  MoveL 642 to (10.69, 196.46, 60) mm, rotated rx -73.66 ry -11.39 rz 28.02 deg; joints [-11.348, -51.869, 112.326, 18.148, -107.646, 15.462, -1511.595]
  MoveL 643 to (4.64, 195.67, 50) mm, rotated rx -73.16 ry -13.02 rz 26.6 deg; joints [-11.489, -49.859, 112.079, 20.024, -113.289, 18.13, -1506.075]
  MoveL 644 to (-1.18, 195.49, 40) mm, rotated rx -74.98 ry -12.29 rz 16.89 deg; joints [-11.645, -52.231, 112.35, 18.85, -106.89, 14.37, -1500.872]
  MoveL 645 to (-6.67, 195.86, 30) mm, rotated rx -74.62 ry -14.16 rz 16.83 deg; joints [-11.702, -49.919, 112.059, 21.112, -113.427, 17.304, -1496.017]
  MoveL 646 to (-11.76, 196.67, 20) mm, rotated rx -76.4 ry -13.89 rz 8.51 deg; joints [-11.758, -51.951, 112.266, 20.461, -107.995, 13.792, -1491.54]
  MoveL 647 to (-16.38, 197.8, 10) mm, rotated rx -78.17 ry -13.98 rz 0.96 deg; joints [-11.742, -53.642, 112.118, 20.427, -102.896, 10.543, -1487.469]
  MoveL 648 to (-20.49, 199.16, 0) mm, rotated rx -78.17 ry -13.98 rz 0.96 deg; joints [-12.168, -53.619, 111.889, 20.096, -102.626, 10.685, -1487.469]
  Set speed (1000.0 mm/s)
  MoveL 649 to (-20.49, 199.16, 0) mm, rotated rx -78.17 ry -13.98 rz 0.96 deg; joints [-12.168, -53.619, 111.889, 20.096, -102.626, 10.685, -1487.469]
  Set speed (1000.0 mm/s)
  MoveL 650 to (37.11, 300.24, 290) mm, rotated rx -90 ry -25 rz -166.45 deg; joints [2.992, -46.004, 98.028, 40.584, -108.594, -7.061, -1313.547]
  MoveL 651 to (37.11, 300.24, 290) mm, rotated rx -90 ry -25 rz -166.45 deg; joints [2.992, -46.004, 98.028, 40.584, -108.594, -7.061, -1313.547]
  Set speed (60.0 mm/s)
  MoveL 652 to (43.85, 319.91, 290) mm, rotated rx -90 ry -25 rz -162.09 deg; joints [2.992, -46.901, 97.924, 40.37, -107.832, -7.745, -1317.907]
  Set speed (1000.0 mm/s)
  MoveL 653 to (43.85, 319.91, 290) mm, rotated rx -90 ry -25 rz -162.09 deg; joints [2.992, -46.901, 97.924, 40.37, -107.832, -7.745, -1317.907]
  Set speed (1000.0 mm/s)
  MoveL 654 to (-20.49, 199.16, 0) mm, rotated rx -90 ry -25 rz 28.05 deg; joints [-7.468, -49.938, 106.45, 34.613, -108.412, 0.917, -1148.047]
  MoveL 655 to (-20.49, 199.16, 0) mm, rotated rx -90 ry -25 rz 28.05 deg; joints [-7.468, -49.938, 106.45, 34.613, -108.412, 0.917, -1148.047]
  Set speed (60.0 mm/s)
  MoveL 656 to (-20.57, 178.36, 0) mm, rotated rx -90 ry -25 rz 33.98 deg; joints [-7.468, -50.9, 106.359, 34.42, -107.545, 0.29, -1153.977]
  Set speed (1000.0 mm/s)
  MoveL 657 to (-20.57, 178.36, 0) mm, rotated rx -90 ry -25 rz 33.98 deg; joints [-7.468, -50.9, 106.359, 34.42, -107.545, 0.29, -1153.977]
  Set speed (1000.0 mm/s)
  MoveL 658 to (-20.49, 199.16, 0) mm, rotated rx -90 ry -25 rz 28.05 deg; joints [-7.468, -49.938, 106.45, 34.613, -108.412, 0.917, -1148.047]
  MoveL 659 to (-20.49, 199.16, 0) mm, rotated rx -90 ry -25 rz 28.05 deg; joints [-7.468, -49.938, 106.45, 34.613, -108.412, 0.917, -1148.047]
  Set speed (60.0 mm/s)
  MoveL 660 to (-16.38, 197.8, 10) mm, rotated rx -90 ry -25 rz 32.58 deg; joints [-7.088, -49.83, 106.249, 34.855, -108.455, 0.679, -1152.579]
  MoveL 661 to (-11.76, 196.67, 20) mm, rotated rx -90 ry -25 rz 37.57 deg; joints [-6.709, -49.719, 106.042, 35.094, -108.496, 0.44, -1157.568]
  MoveL 662 to (-6.67, 195.86, 30) mm, rotated rx -90 ry -25 rz 42.97 deg; joints [-6.332, -49.607, 105.829, 35.331, -108.535, 0.198, -1162.975]
  MoveL 663 to (-1.18, 195.49, 40) mm, rotated rx -90 ry -25 rz 48.76 deg; joints [-5.956, -49.493, 105.609, 35.566, -108.57, -0.047, -1168.76]
  MoveL 664 to (4.64, 195.67, 50) mm, rotated rx -90 ry -25 rz 54.88 deg; joints [-5.581, -49.378, 105.383, 35.798, -108.602, -0.295, -1174.88]
  MoveL 665 to (10.69, 196.46, 60) mm, rotated rx -90 ry -25 rz 61.29 deg; joints [-5.207, -49.263, 105.151, 36.028, -108.63, -0.546, -1181.291]
  MoveL 666 to (16.86, 197.94, 70) mm, rotated rx -90 ry -25 rz 67.95 deg; joints [-4.834, -49.146, 104.912, 36.254, -108.654, -0.801, -1187.947]
  MoveL 667 to (23.03, 200.17, 80) mm, rotated rx -90 ry -25 rz 74.8 deg; joints [-4.463, -49.03, 104.666, 36.478, -108.674, -1.059, -1194.802]
  MoveL 668 to (29.06, 203.14, 90) mm, rotated rx -90 ry -25 rz 81.81 deg; joints [-4.093, -48.913, 104.414, 36.699, -108.69, -1.322, -1201.809]
  MoveL 669 to (34.83, 206.87, 100) mm, rotated rx -90 ry -25 rz 88.92 deg; joints [-3.725, -48.796, 104.156, 36.917, -108.702, -1.588, -1208.92]
  MoveL 670 to (40.19, 211.31, 110) mm, rotated rx -90 ry -25 rz 96.09 deg; joints [-3.358, -48.678, 103.891, 37.133, -108.711, -1.858, -1216.089]
  MoveL 671 to (45.04, 216.4, 120) mm, rotated rx -90 ry -25 rz 103.27 deg; joints [-2.992, -48.56, 103.619, 37.345, -108.716, -2.131, -1223.271]
  MoveL 672 to (49.26, 222.05, 130) mm, rotated rx -90 ry -25 rz 110.42 deg; joints [-2.628, -48.44, 103.341, 37.555, -108.717, -2.408, -1230.424]
  MoveL 673 to (52.77, 228.15, 140) mm, rotated rx -90 ry -25 rz 117.51 deg; joints [-2.265, -48.318, 103.057, 37.761, -108.716, -2.687, -1237.506]
  MoveL 674 to (55.51, 234.59, 150) mm, rotated rx -90 ry -25 rz 124.48 deg; joints [-1.904, -48.193, 102.766, 37.966, -108.713, -2.97, -1244.481]
  MoveL 675 to (57.45, 241.22, 160) mm, rotated rx -90 ry -25 rz 131.31 deg; joints [-1.544, -48.066, 102.469, 38.167, -108.708, -3.254, -1251.311]
  MoveL 676 to (58.59, 247.92, 170) mm, rotated rx -90 ry -25 rz 137.96 deg; joints [-1.185, -47.936, 102.165, 38.366, -108.701, -3.541, -1257.965]
  MoveL 677 to (58.95, 254.55, 180) mm, rotated rx -90 ry -25 rz 144.41 deg; joints [-0.828, -47.802, 101.855, 38.563, -108.694, -3.829, -1264.41]
  MoveL 678 to (58.59, 260.98, 190) mm, rotated rx -90 ry -25 rz 150.62 deg; joints [-0.473, -47.664, 101.539, 38.758, -108.685, -4.119, -1270.617]
  MoveL 679 to (57.57, 267.12, 200) mm, rotated rx -90 ry -25 rz 156.56 deg; joints [-0.119, -47.521, 101.216, 38.95, -108.677, -4.409, -1276.558]
  MoveL 680 to (56, 272.86, 210) mm, rotated rx -90 ry -25 rz 162.2 deg; joints [0.233, -47.373, 100.887, 39.14, -108.668, -4.701, -1282.205]
  MoveL 681 to (53.98, 278.14, 220) mm, rotated rx -90 ry -25 rz 167.53 deg; joints [0.584, -47.22, 100.552, 39.328, -108.659, -4.994, -1287.531]
  MoveL 682 to (51.62, 282.9, 230) mm, rotated rx -90 ry -25 rz 172.51 deg; joints [0.933, -47.062, 100.211, 39.514, -108.65, -5.287, -1292.509]
  MoveL 683 to (49.06, 287.12, 240) mm, rotated rx -90 ry -25 rz 177.11 deg; joints [1.28, -46.898, 99.863, 39.698, -108.641, -5.581, -1297.114]
  MoveL 684 to (46.4, 290.79, 250) mm, rotated rx -90 ry -25 rz -178.68 deg; joints [1.626, -46.729, 99.509, 39.879, -108.632, -5.875, -1301.316]
  MoveL 685 to (43.78, 293.91, 260) mm, rotated rx -90 ry -25 rz -174.91 deg; joints [1.97, -46.556, 99.148, 40.059, -108.623, -6.17, -1305.09]
  MoveL 686 to (41.29, 296.51, 270) mm, rotated rx -90 ry -25 rz -171.59 deg; joints [2.312, -46.377, 98.781, 40.236, -108.614, -6.466, -1308.405]
  MoveL 687 to (39.03, 298.61, 280) mm, rotated rx -90 ry -25 rz -168.77 deg; joints [2.653, -46.193, 98.408, 40.411, -108.604, -6.763, -1311.234]
  MoveL 688 to (37.11, 300.24, 290) mm, rotated rx -90 ry -25 rz -166.45 deg; joints [2.992, -46.004, 98.028, 40.584, -108.594, -7.061, -1313.547]
  Set speed (1000.0 mm/s)
  MoveL 689 to (37.11, 300.24, 290) mm, rotated rx -90 ry -25 rz -166.45 deg; joints [2.992, -46.004, 98.028, 40.584, -108.594, -7.061, -1313.547]
  Set speed (1000.0 mm/s)
  MoveL 690 to (43.85, 319.91, 290) mm, rotated rx -90 ry -25 rz -162.09 deg; joints [2.992, -46.901, 97.924, 40.37, -107.832, -7.745, -1317.907]
  MoveL 691 to (43.85, 319.91, 290) mm, rotated rx -90 ry -25 rz -162.09 deg; joints [2.992, -46.901, 97.924, 40.37, -107.832, -7.745, -1317.907]
  Set speed (60.0 mm/s)
  MoveL 692 to (46.6, 317.98, 280) mm, rotated rx -90 ry -25 rz -164.43 deg; joints [2.653, -47.093, 98.303, 40.197, -107.838, -7.447, -1315.567]
  MoveL 693 to (49.86, 315.46, 270) mm, rotated rx -90 ry -25 rz -167.29 deg; joints [2.312, -47.281, 98.677, 40.022, -107.842, -7.151, -1312.706]
  MoveL 694 to (53.49, 312.31, 260) mm, rotated rx -90 ry -25 rz -170.65 deg; joints [1.97, -47.464, 99.044, 39.845, -107.847, -6.855, -1309.355]
  MoveL 695 to (57.36, 308.47, 250) mm, rotated rx -90 ry -25 rz -174.45 deg; joints [1.626, -47.641, 99.405, 39.665, -107.851, -6.559, -1305.545]
  MoveL 696 to (61.34, 303.9, 240) mm, rotated rx -90 ry -25 rz -178.69 deg; joints [1.28, -47.814, 99.759, 39.484, -107.855, -6.265, -1301.306]
  MoveL 697 to (65.27, 298.59, 230) mm, rotated rx -90 ry -25 rz 176.67 deg; joints [0.933, -47.981, 100.107, 39.3, -107.859, -5.97, -1296.668]
  MoveL 698 to (68.98, 292.54, 220) mm, rotated rx -90 ry -25 rz 171.66 deg; joints [0.584, -48.143, 100.449, 39.114, -107.864, -5.677, -1291.66]
  MoveL 699 to (72.31, 285.76, 210) mm, rotated rx -90 ry -25 rz 166.31 deg; joints [0.233, -48.3, 100.785, 38.926, -107.868, -5.384, -1286.311]
  MoveL 700 to (75.1, 278.3, 200) mm, rotated rx -90 ry -25 rz 160.65 deg; joints [-0.119, -48.452, 101.115, 38.736, -107.872, -5.092, -1280.65]
  MoveL 701 to (77.2, 270.26, 190) mm, rotated rx -90 ry -25 rz 154.71 deg; joints [-0.473, -48.599, 101.438, 38.544, -107.877, -4.8, -1274.706]
  MoveL 702 to (78.47, 261.74, 180) mm, rotated rx -90 ry -25 rz 148.51 deg; joints [-0.828, -48.74, 101.755, 38.35, -107.881, -4.509, -1268.508]
  MoveL 703 to (78.79, 252.87, 170) mm, rotated rx -90 ry -25 rz 142.09 deg; joints [-1.185, -48.878, 102.066, 38.153, -107.884, -4.22, -1262.086]
  MoveL 704 to (78.09, 243.82, 160) mm, rotated rx -90 ry -25 rz 135.47 deg; joints [-1.544, -49.011, 102.37, 37.955, -107.887, -3.932, -1255.472]
  MoveL 705 to (76.31, 234.75, 150) mm, rotated rx -90 ry -25 rz 128.7 deg; joints [-1.904, -49.141, 102.668, 37.753, -107.888, -3.645, -1248.696]
  MoveL 706 to (73.44, 225.85, 140) mm, rotated rx -90 ry -25 rz 121.79 deg; joints [-2.265, -49.268, 102.96, 37.55, -107.888, -3.361, -1241.794]
  MoveL 707 to (69.5, 217.29, 130) mm, rotated rx -90 ry -25 rz 114.8 deg; joints [-2.628, -49.392, 103.245, 37.344, -107.885, -3.079, -1234.8]
  MoveL 708 to (64.57, 209.26, 120) mm, rotated rx -90 ry -25 rz 107.75 deg; joints [-2.992, -49.514, 103.524, 37.135, -107.88, -2.8, -1227.751]
  MoveL 709 to (58.74, 201.9, 110) mm, rotated rx -90 ry -25 rz 100.69 deg; joints [-3.358, -49.634, 103.796, 36.924, -107.872, -2.524, -1220.687]
  MoveL 710 to (52.14, 195.34, 100) mm, rotated rx -90 ry -25 rz 93.65 deg; joints [-3.725, -49.753, 104.062, 36.709, -107.861, -2.251, -1213.646]
  MoveL 711 to (44.91, 189.68, 90) mm, rotated rx -90 ry -25 rz 86.67 deg; joints [-4.093, -49.872, 104.321, 36.492, -107.846, -1.982, -1206.671]
  MoveL 712 to (37.24, 184.98, 80) mm, rotated rx -90 ry -25 rz 79.81 deg; joints [-4.463, -49.989, 104.574, 36.273, -107.827, -1.716, -1199.806]
  MoveL 713 to (29.3, 181.28, 70) mm, rotated rx -90 ry -25 rz 73.09 deg; joints [-4.834, -50.106, 104.82, 36.05, -107.805, -1.454, -1193.092]
  MoveL 714 to (21.27, 178.55, 60) mm, rotated rx -90 ry -25 rz 66.58 deg; joints [-5.207, -50.223, 105.059, 35.825, -107.778, -1.196, -1186.575]
  MoveL 715 to (13.31, 176.76, 50) mm, rotated rx -90 ry -25 rz 60.3 deg; joints [-5.581, -50.339, 105.292, 35.597, -107.748, -0.941, -1180.298]
  MoveL 716 to (5.58, 175.83, 40) mm, rotated rx -90 ry -25 rz 54.3 deg; joints [-5.956, -50.454, 105.518, 35.366, -107.714, -0.689, -1174.303]
  MoveL 717 to (-1.77, 175.65, 30) mm, rotated rx -90 ry -25 rz 48.63 deg; joints [-6.332, -50.568, 105.738, 35.133, -107.676, -0.44, -1168.634]
  MoveL 718 to (-8.64, 176.1, 20) mm, rotated rx -90 ry -25 rz 43.33 deg; joints [-6.709, -50.68, 105.952, 34.897, -107.635, -0.195, -1163.33]
  MoveL 719 to (-14.93, 177.06, 10) mm, rotated rx -90 ry -25 rz 38.43 deg; joints [-7.088, -50.791, 106.159, 34.66, -107.591, 0.049, -1158.431]
  MoveL 720 to (-20.57, 178.36, 0) mm, rotated rx -90 ry -25 rz 33.98 deg; joints [-7.468, -50.9, 106.359, 34.42, -107.545, 0.29, -1153.977]
  Set speed (1000.0 mm/s)
  MoveL 721 to (-20.57, 178.36, 0) mm, rotated rx -90 ry -25 rz 33.98 deg; joints [-7.468, -50.9, 106.359, 34.42, -107.545, 0.29, -1153.977]
  Set speed (1000.0 mm/s)
  MoveL 722 to (43.85, 319.91, 290) mm, rotated rx -90 ry -25 rz -162.09 deg; joints [2.992, -46.901, 97.924, 40.37, -107.832, -7.745, -1317.907]
  MoveL 723 to (43.85, 319.91, 290) mm, rotated rx -90 ry -25 rz -162.09 deg; joints [2.992, -46.901, 97.924, 40.37, -107.832, -7.745, -1317.907]
  Set speed (60.0 mm/s)
  MoveL 724 to (28.22, 306.19, 290) mm, rotated rx -90 ry -25 rz -156.66 deg; joints [2.992, -46.023, 98.026, 40.579, -108.578, -7.075, -1323.337]
  Set speed (1000.0 mm/s)
  MoveL 725 to (28.22, 306.19, 290) mm, rotated rx -90 ry -25 rz -156.66 deg; joints [2.992, -46.023, 98.026, 40.579, -108.578, -7.075, -1323.337]
  Set speed (1000.0 mm/s)
  MoveL 726 to (-20.57, 178.36, 0) mm, rotated rx -90 ry -25 rz 33.98 deg; joints [-7.468, -50.9, 106.359, 34.42, -107.545, 0.29, -1153.977]
  MoveL 727 to (-20.57, 178.36, 0) mm, rotated rx -90 ry -25 rz 33.98 deg; joints [-7.468, -50.9, 106.359, 34.42, -107.545, 0.29, -1153.977]
  Set speed (60.0 mm/s)
  MoveL 728 to (-10.16, 196.36, 0) mm, rotated rx -90 ry -25 rz 39.27 deg; joints [-7.468, -49.927, 106.451, 34.616, -108.422, 0.924, -1159.273]
  Set speed (1000.0 mm/s)
  MoveL 729 to (-10.16, 196.36, 0) mm, rotated rx -90 ry -25 rz 39.27 deg; joints [-7.468, -49.927, 106.451, 34.616, -108.422, 0.924, -1159.273]
  Set speed (1000.0 mm/s)
  MoveL 730 to (-20.57, 178.36, 0) mm, rotated rx -90 ry -25 rz 33.98 deg; joints [-7.468, -50.9, 106.359, 34.42, -107.545, 0.29, -1153.977]
  MoveL 731 to (-20.57, 178.36, 0) mm, rotated rx -90 ry -25 rz 33.98 deg; joints [-7.468, -50.9, 106.359, 34.42, -107.545, 0.29, -1153.977]
  Set speed (60.0 mm/s)
  MoveL 732 to (-14.93, 177.06, 10) mm, rotated rx -90 ry -25 rz 38.43 deg; joints [-7.088, -50.791, 106.159, 34.66, -107.591, 0.049, -1158.431]
  MoveL 733 to (-8.64, 176.1, 20) mm, rotated rx -90 ry -25 rz 43.33 deg; joints [-6.709, -50.68, 105.952, 34.897, -107.635, -0.195, -1163.33]
  MoveL 734 to (-1.77, 175.65, 30) mm, rotated rx -90 ry -25 rz 48.63 deg; joints [-6.332, -50.568, 105.738, 35.133, -107.676, -0.44, -1168.634]
  MoveL 735 to (5.58, 175.83, 40) mm, rotated rx -90 ry -25 rz 54.3 deg; joints [-5.956, -50.454, 105.518, 35.366, -107.714, -0.689, -1174.303]
  MoveL 736 to (13.31, 176.76, 50) mm, rotated rx -90 ry -25 rz 60.3 deg; joints [-5.581, -50.339, 105.292, 35.597, -107.748, -0.941, -1180.298]
  MoveL 737 to (21.27, 178.55, 60) mm, rotated rx -90 ry -25 rz 66.58 deg; joints [-5.207, -50.223, 105.059, 35.825, -107.778, -1.196, -1186.575]
  MoveL 738 to (29.3, 181.28, 70) mm, rotated rx -90 ry -25 rz 73.09 deg; joints [-4.834, -50.106, 104.82, 36.05, -107.805, -1.454, -1193.092]
  MoveL 739 to (37.24, 184.98, 80) mm, rotated rx -90 ry -25 rz 79.81 deg; joints [-4.463, -49.989, 104.574, 36.273, -107.827, -1.716, -1199.806]
  MoveL 740 to (44.91, 189.68, 90) mm, rotated rx -90 ry -25 rz 86.67 deg; joints [-4.093, -49.872, 104.321, 36.492, -107.846, -1.982, -1206.671]
  MoveL 741 to (52.14, 195.34, 100) mm, rotated rx -90 ry -25 rz 93.65 deg; joints [-3.725, -49.753, 104.062, 36.709, -107.861, -2.251, -1213.646]
  MoveL 742 to (58.74, 201.9, 110) mm, rotated rx -90 ry -25 rz 100.69 deg; joints [-3.358, -49.634, 103.796, 36.924, -107.872, -2.524, -1220.687]
  MoveL 743 to (64.57, 209.26, 120) mm, rotated rx -90 ry -25 rz 107.75 deg; joints [-2.992, -49.514, 103.524, 37.135, -107.88, -2.8, -1227.751]
  MoveL 744 to (69.5, 217.29, 130) mm, rotated rx -90 ry -25 rz 114.8 deg; joints [-2.628, -49.392, 103.245, 37.344, -107.885, -3.079, -1234.8]
  MoveL 745 to (73.44, 225.85, 140) mm, rotated rx -90 ry -25 rz 121.79 deg; joints [-2.265, -49.268, 102.96, 37.55, -107.888, -3.361, -1241.794]
  MoveL 746 to (76.31, 234.75, 150) mm, rotated rx -90 ry -25 rz 128.7 deg; joints [-1.904, -49.141, 102.668, 37.753, -107.888, -3.645, -1248.696]
  MoveL 747 to (78.09, 243.82, 160) mm, rotated rx -90 ry -25 rz 135.47 deg; joints [-1.544, -49.011, 102.37, 37.955, -107.887, -3.932, -1255.472]
  MoveL 748 to (78.79, 252.87, 170) mm, rotated rx -90 ry -25 rz 142.09 deg; joints [-1.185, -48.878, 102.066, 38.153, -107.884, -4.22, -1262.086]
  MoveL 749 to (78.47, 261.74, 180) mm, rotated rx -90 ry -25 rz 148.51 deg; joints [-0.828, -48.74, 101.755, 38.35, -107.881, -4.509, -1268.508]
  MoveL 750 to (77.2, 270.26, 190) mm, rotated rx -90 ry -25 rz 154.71 deg; joints [-0.473, -48.599, 101.438, 38.544, -107.877, -4.8, -1274.706]
  MoveL 751 to (75.1, 278.3, 200) mm, rotated rx -90 ry -25 rz 160.65 deg; joints [-0.119, -48.452, 101.115, 38.736, -107.872, -5.092, -1280.65]
  MoveL 752 to (72.31, 285.76, 210) mm, rotated rx -90 ry -25 rz 166.31 deg; joints [0.233, -48.3, 100.785, 38.926, -107.868, -5.384, -1286.311]
  MoveL 753 to (68.98, 292.54, 220) mm, rotated rx -90 ry -25 rz 171.66 deg; joints [0.584, -48.143, 100.449, 39.114, -107.864, -5.677, -1291.66]
  MoveL 754 to (65.27, 298.59, 230) mm, rotated rx -90 ry -25 rz 176.67 deg; joints [0.933, -47.981, 100.107, 39.3, -107.859, -5.97, -1296.668]
  MoveL 755 to (61.34, 303.9, 240) mm, rotated rx -90 ry -25 rz -178.69 deg; joints [1.28, -47.814, 99.759, 39.484, -107.855, -6.265, -1301.306]
  MoveL 756 to (57.36, 308.47, 250) mm, rotated rx -90 ry -25 rz -174.45 deg; joints [1.626, -47.641, 99.405, 39.665, -107.851, -6.559, -1305.545]
  MoveL 757 to (53.49, 312.31, 260) mm, rotated rx -90 ry -25 rz -170.65 deg; joints [1.97, -47.464, 99.044, 39.845, -107.847, -6.855, -1309.355]
  MoveL 758 to (49.86, 315.46, 270) mm, rotated rx -90 ry -25 rz -167.29 deg; joints [2.312, -47.281, 98.677, 40.022, -107.842, -7.151, -1312.706]
  MoveL 759 to (46.6, 317.98, 280) mm, rotated rx -90 ry -25 rz -164.43 deg; joints [2.653, -47.093, 98.303, 40.197, -107.838, -7.447, -1315.567]
  MoveL 760 to (43.85, 319.91, 290) mm, rotated rx -90 ry -25 rz -162.09 deg; joints [2.992, -46.901, 97.924, 40.37, -107.832, -7.745, -1317.907]
  Set speed (1000.0 mm/s)
  MoveL 761 to (43.85, 319.91, 290) mm, rotated rx -90 ry -25 rz -162.09 deg; joints [2.992, -46.901, 97.924, 40.37, -107.832, -7.745, -1317.907]
  Set speed (1000.0 mm/s)
  MoveL 762 to (28.22, 306.19, 290) mm, rotated rx -90 ry -25 rz -156.66 deg; joints [2.992, -46.023, 98.026, 40.579, -108.578, -7.075, -1323.337]
  MoveL 763 to (28.22, 306.19, 290) mm, rotated rx -90 ry -25 rz -156.66 deg; joints [2.992, -46.023, 98.026, 40.579, -108.578, -7.075, -1323.337]
  Set speed (60.0 mm/s)
  MoveL 764 to (30.4, 304.94, 280) mm, rotated rx -90 ry -25 rz -158.96 deg; joints [2.653, -46.213, 98.406, 40.406, -108.587, -6.778, -1321.04]
  MoveL 765 to (33, 303.28, 270) mm, rotated rx -90 ry -25 rz -161.77 deg; joints [2.312, -46.398, 98.779, 40.231, -108.595, -6.483, -1318.23]
  MoveL 766 to (35.92, 301.18, 260) mm, rotated rx -90 ry -25 rz -165.06 deg; joints [1.97, -46.579, 99.146, 40.053, -108.603, -6.188, -1314.94]
  MoveL 767 to (39.07, 298.58, 250) mm, rotated rx -90 ry -25 rz -168.8 deg; joints [1.626, -46.755, 99.506, 39.873, -108.61, -5.894, -1311.197]
  MoveL 768 to (42.34, 295.45, 240) mm, rotated rx -90 ry -25 rz -172.97 deg; joints [1.28, -46.926, 99.86, 39.691, -108.618, -5.601, -1307.031]
  MoveL 769 to (45.62, 291.76, 230) mm, rotated rx -90 ry -25 rz -177.53 deg; joints [0.933, -47.091, 100.208, 39.507, -108.625, -5.308, -1302.471]
  MoveL 770 to (48.8, 287.5, 220) mm, rotated rx -90 ry -25 rz 177.54 deg; joints [0.584, -47.251, 100.549, 39.321, -108.632, -5.016, -1297.543]
  MoveL 771 to (51.74, 282.68, 210) mm, rotated rx -90 ry -25 rz 172.28 deg; joints [0.233, -47.406, 100.884, 39.133, -108.64, -4.725, -1292.275]
  MoveL 772 to (54.33, 277.32, 200) mm, rotated rx -90 ry -25 rz 166.69 deg; joints [-0.119, -47.555, 101.213, 38.942, -108.647, -4.435, -1286.694]
  MoveL 773 to (56.44, 271.47, 190) mm, rotated rx -90 ry -25 rz 160.83 deg; joints [-0.473, -47.7, 101.535, 38.75, -108.655, -4.145, -1280.826]
  MoveL 774 to (57.96, 265.2, 180) mm, rotated rx -90 ry -25 rz 154.7 deg; joints [-0.828, -47.839, 101.852, 38.555, -108.662, -3.856, -1274.699]
  MoveL 775 to (58.8, 258.62, 170) mm, rotated rx -90 ry -25 rz 148.34 deg; joints [-1.185, -47.974, 102.162, 38.358, -108.669, -3.568, -1268.339]
  MoveL 776 to (58.89, 251.83, 160) mm, rotated rx -90 ry -25 rz 141.78 deg; joints [-1.544, -48.104, 102.465, 38.159, -108.676, -3.281, -1261.776]
  MoveL 777 to (58.18, 244.95, 150) mm, rotated rx -90 ry -25 rz 135.04 deg; joints [-1.904, -48.231, 102.763, 37.957, -108.681, -2.996, -1255.039]
  MoveL 778 to (56.65, 238.12, 140) mm, rotated rx -90 ry -25 rz 128.16 deg; joints [-2.265, -48.354, 103.054, 37.753, -108.685, -2.713, -1248.16]
  MoveL 779 to (54.3, 231.49, 130) mm, rotated rx -90 ry -25 rz 121.17 deg; joints [-2.628, -48.474, 103.338, 37.547, -108.687, -2.432, -1241.173]
  MoveL 780 to (51.17, 225.17, 120) mm, rotated rx -90 ry -25 rz 114.11 deg; joints [-2.992, -48.592, 103.616, 37.338, -108.687, -2.154, -1234.112]
  MoveL 781 to (47.33, 219.29, 110) mm, rotated rx -90 ry -25 rz 107.02 deg; joints [-3.358, -48.708, 103.888, 37.126, -108.685, -1.879, -1227.017]
  MoveL 782 to (42.85, 213.95, 100) mm, rotated rx -90 ry -25 rz 99.93 deg; joints [-3.725, -48.823, 104.153, 36.911, -108.679, -1.606, -1219.928]
  MoveL 783 to (37.86, 209.24, 90) mm, rotated rx -90 ry -25 rz 92.89 deg; joints [-4.093, -48.937, 104.412, 36.694, -108.67, -1.338, -1212.888]
  MoveL 784 to (32.46, 205.23, 80) mm, rotated rx -90 ry -25 rz 85.94 deg; joints [-4.463, -49.05, 104.664, 36.474, -108.657, -1.073, -1205.942]
  MoveL 785 to (26.8, 201.92, 70) mm, rotated rx -90 ry -25 rz 79.14 deg; joints [-4.834, -49.162, 104.91, 36.251, -108.64, -0.811, -1199.135]
  MoveL 786 to (21, 199.35, 60) mm, rotated rx -90 ry -25 rz 72.51 deg; joints [-5.207, -49.274, 105.15, 36.025, -108.62, -0.554, -1192.515]
  MoveL 787 to (15.19, 197.47, 50) mm, rotated rx -90 ry -25 rz 66.13 deg; joints [-5.581, -49.385, 105.383, 35.797, -108.596, -0.3, -1186.127]
  MoveL 788 to (9.5, 196.25, 40) mm, rotated rx -90 ry -25 rz 60.02 deg; joints [-5.956, -49.496, 105.609, 35.565, -108.567, -0.049, -1180.02]
  MoveL 789 to (4.03, 195.62, 30) mm, rotated rx -90 ry -25 rz 54.24 deg; joints [-6.332, -49.606, 105.829, 35.332, -108.536, 0.199, -1174.238]
  MoveL 790 to (-1.12, 195.49, 20) mm, rotated rx -90 ry -25 rz 48.82 deg; joints [-6.709, -49.715, 106.043, 35.095, -108.501, 0.443, -1168.824]
  MoveL 791 to (-5.87, 195.78, 10) mm, rotated rx -90 ry -25 rz 43.82 deg; joints [-7.088, -49.822, 106.25, 34.856, -108.462, 0.685, -1163.823]
  MoveL 792 to (-10.16, 196.36, 0) mm, rotated rx -90 ry -25 rz 39.27 deg; joints [-7.468, -49.927, 106.451, 34.616, -108.422, 0.924, -1159.273]
  Set speed (1000.0 mm/s)
  MoveL 793 to (-10.16, 196.36, 0) mm, rotated rx -90 ry -25 rz 39.27 deg; joints [-7.468, -49.927, 106.451, 34.616, -108.422, 0.924, -1159.273]
  Set speed (1000.0 mm/s)
  MoveL 794 to (28.22, 306.19, 290) mm, rotated rx -90 ry -25 rz -156.66 deg; joints [2.992, -46.023, 98.026, 40.579, -108.578, -7.075, -1323.337]
  MoveL 795 to (28.22, 306.19, 290) mm, rotated rx -90 ry -25 rz -156.66 deg; joints [2.992, -46.023, 98.026, 40.579, -108.578, -7.075, -1323.337]
  Set speed (60.0 mm/s)
  MoveL 796 to (-21.11, 309.47, 290) mm, rotated rx -90 ry -25 rz -110.46 deg; joints [2.992, -46.033, 98.025, 40.576, -108.57, -7.083, -1369.544]
  Set speed (1000.0 mm/s)
  MoveL 797 to (-21.11, 309.47, 290) mm, rotated rx -90 ry -25 rz -110.46 deg; joints [2.992, -46.033, 98.025, 40.576, -108.57, -7.083, -1369.544]
  Set speed (1000.0 mm/s)
  MoveL 798 to (-10.16, 196.36, 0) mm, rotated rx -90 ry -25 rz 39.27 deg; joints [-7.468, -49.927, 106.451, 34.616, -108.422, 0.924, -1519.273]
  MoveL 799 to (-10.16, 196.36, 0) mm, rotated rx -90 ry -25 rz 39.27 deg; joints [-7.468, -49.927, 106.451, 34.616, -108.422, 0.924, -1519.273]
  Set speed (60.0 mm/s)
  MoveL 800 to (37.62, 209.05, 0) mm, rotated rx -90 ry -25 rz 92.57 deg; joints [-7.468, -49.977, 106.447, 34.605, -108.377, 0.891, -1572.574]
  Set speed (1000.0 mm/s)
  MoveL 801 to (37.62, 209.05, 0) mm, rotated rx -90 ry -25 rz 92.57 deg; joints [-7.468, -49.977, 106.447, 34.605, -108.377, 0.891, -1572.574]
  Set speed (1000.0 mm/s)
  MoveL 802 to (-10.16, 196.36, 0) mm, rotated rx -90 ry -25 rz 39.27 deg; joints [-7.468, -49.927, 106.451, 34.616, -108.422, 0.924, -1519.273]
  MoveL 803 to (-10.16, 196.36, 0) mm, rotated rx -90 ry -25 rz 39.27 deg; joints [-7.468, -49.927, 106.451, 34.616, -108.422, 0.924, -1519.273]
  Set speed (60.0 mm/s)
  MoveL 804 to (-5.87, 195.78, 10) mm, rotated rx -90 ry -25 rz 43.82 deg; joints [-7.088, -49.822, 106.25, 34.856, -108.462, 0.685, -1523.823]
  MoveL 805 to (-1.12, 195.49, 20) mm, rotated rx -90 ry -25 rz 48.82 deg; joints [-6.709, -49.715, 106.043, 35.095, -108.501, 0.443, -1528.824]
  MoveL 806 to (4.03, 195.62, 30) mm, rotated rx -90 ry -25 rz 54.24 deg; joints [-6.332, -49.606, 105.829, 35.332, -108.536, 0.199, -1534.238]
  MoveL 807 to (9.5, 196.25, 40) mm, rotated rx -90 ry -25 rz 60.02 deg; joints [-5.956, -49.496, 105.609, 35.565, -108.567, -0.049, -1540.02]
  MoveL 808 to (15.19, 197.47, 50) mm, rotated rx -90 ry -25 rz 66.13 deg; joints [-5.581, -49.385, 105.383, 35.797, -108.596, -0.3, -1546.127]
  MoveL 809 to (21, 199.35, 60) mm, rotated rx -90 ry -25 rz 72.51 deg; joints [-5.207, -49.274, 105.15, 36.025, -108.62, -0.554, -1552.515]
  MoveL 810 to (26.8, 201.92, 70) mm, rotated rx -90 ry -25 rz 79.14 deg; joints [-4.834, -49.162, 104.91, 36.251, -108.64, -0.811, -1559.135]
  MoveL 811 to (32.46, 205.23, 80) mm, rotated rx -90 ry -25 rz 85.94 deg; joints [-4.463, -49.05, 104.664, 36.474, -108.657, -1.073, -1565.942]
  MoveL 812 to (37.86, 209.24, 90) mm, rotated rx -90 ry -25 rz 92.89 deg; joints [-4.093, -48.937, 104.412, 36.694, -108.67, -1.338, -1572.888]
  MoveL 813 to (42.85, 213.95, 100) mm, rotated rx -90 ry -25 rz 99.93 deg; joints [-3.725, -48.823, 104.153, 36.911, -108.679, -1.606, -1579.928]
  MoveL 814 to (47.33, 219.29, 110) mm, rotated rx -90 ry -25 rz 107.02 deg; joints [-3.358, -48.708, 103.888, 37.126, -108.685, -1.879, -1587.017]
  MoveL 815 to (51.17, 225.17, 120) mm, rotated rx -90 ry -25 rz 114.11 deg; joints [-2.992, -48.592, 103.616, 37.338, -108.687, -2.154, -1594.112]
  MoveL 816 to (54.3, 231.49, 130) mm, rotated rx -90 ry -25 rz 121.17 deg; joints [-2.628, -48.474, 103.338, 37.547, -108.687, -2.432, -1601.173]
  MoveL 817 to (56.65, 238.12, 140) mm, rotated rx -90 ry -25 rz 128.16 deg; joints [-2.265, -48.354, 103.054, 37.753, -108.685, -2.713, -1608.16]
  MoveL 818 to (58.18, 244.95, 150) mm, rotated rx -90 ry -25 rz 135.04 deg; joints [-1.904, -48.231, 102.763, 37.957, -108.681, -2.996, -1615.039]
  MoveL 819 to (58.89, 251.83, 160) mm, rotated rx -90 ry -25 rz 141.78 deg; joints [-1.544, -48.104, 102.465, 38.159, -108.676, -3.281, -1621.776]
  MoveL 820 to (58.8, 258.62, 170) mm, rotated rx -90 ry -25 rz 148.34 deg; joints [-1.185, -47.974, 102.162, 38.358, -108.669, -3.568, -1628.339]
  MoveL 821 to (57.96, 265.2, 180) mm, rotated rx -90 ry -25 rz 154.7 deg; joints [-0.828, -47.839, 101.852, 38.555, -108.662, -3.856, -1634.699]
  MoveL 822 to (56.44, 271.47, 190) mm, rotated rx -90 ry -25 rz 160.83 deg; joints [-0.473, -47.7, 101.535, 38.75, -108.655, -4.145, -1640.826]
  MoveL 823 to (54.33, 277.32, 200) mm, rotated rx -90 ry -25 rz 166.69 deg; joints [-0.119, -47.555, 101.213, 38.942, -108.647, -4.435, -1646.694]
  MoveL 824 to (51.74, 282.68, 210) mm, rotated rx -90 ry -25 rz 172.28 deg; joints [0.233, -47.406, 100.884, 39.133, -108.64, -4.725, -1652.275]
  MoveL 825 to (48.8, 287.5, 220) mm, rotated rx -90 ry -25 rz 177.54 deg; joints [0.584, -47.251, 100.549, 39.321, -108.632, -5.016, -1657.543]
  MoveL 826 to (45.62, 291.76, 230) mm, rotated rx -90 ry -25 rz -177.53 deg; joints [0.933, -47.091, 100.208, 39.507, -108.625, -5.308, -1662.471]
  MoveL 827 to (42.34, 295.45, 240) mm, rotated rx -90 ry -25 rz -172.97 deg; joints [1.28, -46.926, 99.86, 39.691, -108.618, -5.601, -1667.031]
  MoveL 828 to (39.07, 298.58, 250) mm, rotated rx -90 ry -25 rz -168.8 deg; joints [1.626, -46.755, 99.506, 39.873, -108.61, -5.894, -1671.197]
  MoveL 829 to (35.92, 301.18, 260) mm, rotated rx -90 ry -25 rz -165.06 deg; joints [1.97, -46.579, 99.146, 40.053, -108.603, -6.188, -1674.94]
  MoveL 830 to (33, 303.28, 270) mm, rotated rx -90 ry -25 rz -161.77 deg; joints [2.312, -46.398, 98.779, 40.231, -108.595, -6.483, -1678.23]
  MoveL 831 to (30.4, 304.94, 280) mm, rotated rx -90 ry -25 rz -158.96 deg; joints [2.653, -46.213, 98.406, 40.406, -108.587, -6.778, -1681.04]
  MoveL 832 to (28.22, 306.19, 290) mm, rotated rx -90 ry -25 rz -156.66 deg; joints [2.992, -46.023, 98.026, 40.579, -108.578, -7.075, -1683.337]
  Set speed (1000.0 mm/s)
  MoveL 833 to (28.22, 306.19, 290) mm, rotated rx -90 ry -25 rz -156.66 deg; joints [2.992, -46.023, 98.026, 40.579, -108.578, -7.075, -1683.337]
  Set speed (1000.0 mm/s)
  MoveL 834 to (-21.11, 309.47, 290) mm, rotated rx -90 ry -25 rz -110.46 deg; joints [2.992, -46.033, 98.025, 40.576, -108.57, -7.083, -1729.544]
  MoveL 835 to (-21.11, 309.47, 290) mm, rotated rx -90 ry -25 rz -110.46 deg; joints [2.992, -46.033, 98.025, 40.576, -108.57, -7.083, -1729.544]
  Set speed (60.0 mm/s)
  MoveL 836 to (-18.74, 310.33, 280) mm, rotated rx -90 ry -25 rz -112.74 deg; joints [2.653, -46.23, 98.404, 40.402, -108.573, -6.791, -1727.257]
  MoveL 837 to (-15.8, 311.23, 270) mm, rotated rx -90 ry -25 rz -115.53 deg; joints [2.312, -46.424, 98.777, 40.225, -108.574, -6.502, -1724.467]
  MoveL 838 to (-12.3, 312.09, 260) mm, rotated rx -90 ry -25 rz -118.79 deg; joints [1.97, -46.614, 99.142, 40.045, -108.574, -6.214, -1721.209]
  MoveL 839 to (-8.28, 312.8, 250) mm, rotated rx -90 ry -25 rz -122.48 deg; joints [1.626, -46.801, 99.502, 39.863, -108.572, -5.928, -1717.515]
  MoveL 840 to (-3.78, 313.26, 240) mm, rotated rx -90 ry -25 rz -126.58 deg; joints [1.28, -46.983, 99.855, 39.678, -108.569, -5.643, -1713.419]
  MoveL 841 to (1.16, 313.37, 230) mm, rotated rx -90 ry -25 rz -131.05 deg; joints [0.933, -47.161, 100.201, 39.491, -108.565, -5.36, -1708.952]
  MoveL 842 to (6.46, 313.03, 220) mm, rotated rx -90 ry -25 rz -135.85 deg; joints [0.584, -47.335, 100.541, 39.301, -108.561, -5.078, -1704.147]
  MoveL 843 to (12.04, 312.14, 210) mm, rotated rx -90 ry -25 rz -140.97 deg; joints [0.233, -47.503, 100.875, 39.11, -108.557, -4.796, -1699.032]
  MoveL 844 to (17.8, 310.63, 200) mm, rotated rx -90 ry -25 rz -146.36 deg; joints [-0.119, -47.666, 101.203, 38.916, -108.553, -4.515, -1693.638]
  MoveL 845 to (23.62, 308.44, 190) mm, rotated rx -90 ry -25 rz -152.01 deg; joints [-0.473, -47.824, 101.524, 38.721, -108.549, -4.234, -1687.993]
  MoveL 846 to (29.38, 305.54, 180) mm, rotated rx -90 ry -25 rz -157.88 deg; joints [-0.828, -47.975, 101.839, 38.524, -108.546, -3.953, -1682.125]
  MoveL 847 to (34.94, 301.92, 170) mm, rotated rx -90 ry -25 rz -163.94 deg; joints [-1.185, -48.122, 102.148, 38.324, -108.543, -3.673, -1676.061]
  MoveL 848 to (40.17, 297.58, 160) mm, rotated rx -90 ry -25 rz -170.17 deg; joints [-1.544, -48.262, 102.451, 38.123, -108.54, -3.393, -1669.829]
  MoveL 849 to (44.94, 292.58, 150) mm, rotated rx -90 ry -25 rz -176.55 deg; joints [-1.904, -48.397, 102.748, 37.92, -108.539, -3.113, -1663.455]
  MoveL 850 to (49.15, 286.99, 140) mm, rotated rx -90 ry -25 rz 176.97 deg; joints [-2.265, -48.526, 103.038, 37.715, -108.537, -2.834, -1656.967]
  MoveL 851 to (52.68, 280.9, 130) mm, rotated rx -90 ry -25 rz 170.39 deg; joints [-2.628, -48.65, 103.323, 37.508, -108.536, -2.555, -1650.393]
  MoveL 852 to (55.46, 274.42, 120) mm, rotated rx -90 ry -25 rz 163.76 deg; joints [-2.992, -48.77, 103.601, 37.298, -108.534, -2.277, -1643.762]
  MoveL 853 to (57.44, 267.68, 110) mm, rotated rx -90 ry -25 rz 157.1 deg; joints [-3.358, -48.885, 103.873, 37.087, -108.532, -2, -1637.105]
  MoveL 854 to (58.6, 260.81, 100) mm, rotated rx -90 ry -25 rz 150.45 deg; joints [-3.725, -48.996, 104.139, 36.874, -108.529, -1.725, -1630.453]
  MoveL 855 to (58.95, 253.96, 90) mm, rotated rx -90 ry -25 rz 143.84 deg; joints [-4.093, -49.103, 104.398, 36.658, -108.525, -1.451, -1623.84]
  MoveL 856 to (58.51, 247.24, 80) mm, rotated rx -90 ry -25 rz 137.3 deg; joints [-4.463, -49.207, 104.652, 36.44, -108.52, -1.18, -1617.303]
  MoveL 857 to (57.35, 240.79, 70) mm, rotated rx -90 ry -25 rz 130.88 deg; joints [-4.834, -49.309, 104.898, 36.219, -108.512, -0.911, -1610.878]
  MoveL 858 to (55.55, 234.7, 60) mm, rotated rx -90 ry -25 rz 124.6 deg; joints [-5.207, -49.409, 105.139, 35.996, -108.502, -0.644, -1604.605]
  MoveL 859 to (53.21, 229.07, 50) mm, rotated rx -90 ry -25 rz 118.53 deg; joints [-5.581, -49.507, 105.373, 35.771, -108.489, -0.381, -1598.526]
  MoveL 860 to (50.45, 223.94, 40) mm, rotated rx -90 ry -25 rz 112.68 deg; joints [-5.956, -49.603, 105.601, 35.543, -108.473, -0.12, -1592.684]
  MoveL 861 to (47.39, 219.37, 30) mm, rotated rx -90 ry -25 rz 107.12 deg; joints [-6.332, -49.699, 105.822, 35.312, -108.454, 0.138, -1587.123]
  MoveL 862 to (44.15, 215.37, 20) mm, rotated rx -90 ry -25 rz 101.89 deg; joints [-6.709, -49.793, 106.037, 35.079, -108.432, 0.392, -1581.887]
  MoveL 863 to (40.85, 211.93, 10) mm, rotated rx -90 ry -25 rz 97.02 deg; joints [-7.088, -49.886, 106.245, 34.843, -108.406, 0.643, -1577.023]
  MoveL 864 to (37.62, 209.05, 0) mm, rotated rx -90 ry -25 rz 92.57 deg; joints [-7.468, -49.977, 106.447, 34.605, -108.377, 0.891, -1572.574]
  Set speed (1000.0 mm/s)
  MoveL 865 to (37.62, 209.05, 0) mm, rotated rx -90 ry -25 rz 92.57 deg; joints [-7.468, -49.977, 106.447, 34.605, -108.377, 0.891, -1572.574]
  Set speed (1000.0 mm/s)
  MoveL 866 to (-21.11, 309.47, 290) mm, rotated rx -90 ry -25 rz -110.46 deg; joints [2.992, -46.033, 98.025, 40.576, -108.57, -7.083, -1729.544]
  MoveL 867 to (-21.11, 309.47, 290) mm, rotated rx -90 ry -25 rz -110.46 deg; joints [2.992, -46.033, 98.025, 40.576, -108.57, -7.083, -1729.544]
  Set speed (60.0 mm/s)
  MoveL 868 to (-34.79, 325.15, 290) mm, rotated rx -90 ry -25 rz -105.16 deg; joints [2.992, -46.913, 97.922, 40.367, -107.822, -7.755, -1734.84]
  Set speed (1000.0 mm/s)
  MoveL 869 to (-34.79, 325.15, 290) mm, rotated rx -90 ry -25 rz -105.16 deg; joints [2.992, -46.913, 97.922, 40.367, -107.822, -7.755, -1734.84]
  Set speed (1000.0 mm/s)
  MoveL 870 to (37.62, 209.05, 0) mm, rotated rx -90 ry -25 rz 92.57 deg; joints [-7.468, -49.977, 106.447, 34.605, -108.377, 0.891, -1572.574]
  MoveL 871 to (37.62, 209.05, 0) mm, rotated rx -90 ry -25 rz 92.57 deg; joints [-7.468, -49.977, 106.447, 34.605, -108.377, 0.891, -1572.574]
  Set speed (60.0 mm/s)
  MoveL 872 to (55.59, 198.58, 0) mm, rotated rx -90 ry -25 rz 97.23 deg; joints [-7.468, -50.957, 106.353, 34.408, -107.492, 0.252, -1577.234]
  Set speed (1000.0 mm/s)
  MoveL 873 to (55.59, 198.58, 0) mm, rotated rx -90 ry -25 rz 97.23 deg; joints [-7.468, -50.957, 106.353, 34.408, -107.492, 0.252, -1577.234]
  Set speed (1000.0 mm/s)
  MoveL 874 to (37.62, 209.05, 0) mm, rotated rx -90 ry -25 rz 92.57 deg; joints [-7.468, -49.977, 106.447, 34.605, -108.377, 0.891, -1572.574]
  MoveL 875 to (37.62, 209.05, 0) mm, rotated rx -90 ry -25 rz 92.57 deg; joints [-7.468, -49.977, 106.447, 34.605, -108.377, 0.891, -1572.574]
  Set speed (60.0 mm/s)
  MoveL 876 to (40.85, 211.93, 10) mm, rotated rx -90 ry -25 rz 97.02 deg; joints [-7.088, -49.886, 106.245, 34.843, -108.406, 0.643, -1577.023]
  MoveL 877 to (44.15, 215.37, 20) mm, rotated rx -90 ry -25 rz 101.89 deg; joints [-6.709, -49.793, 106.037, 35.079, -108.432, 0.392, -1581.887]
  MoveL 878 to (47.39, 219.37, 30) mm, rotated rx -90 ry -25 rz 107.12 deg; joints [-6.332, -49.699, 105.822, 35.312, -108.454, 0.138, -1587.123]
  MoveL 879 to (50.45, 223.94, 40) mm, rotated rx -90 ry -25 rz 112.68 deg; joints [-5.956, -49.603, 105.601, 35.543, -108.473, -0.12, -1592.684]
  MoveL 880 to (53.21, 229.07, 50) mm, rotated rx -90 ry -25 rz 118.53 deg; joints [-5.581, -49.507, 105.373, 35.771, -108.489, -0.381, -1598.526]
  MoveL 881 to (55.55, 234.7, 60) mm, rotated rx -90 ry -25 rz 124.6 deg; joints [-5.207, -49.409, 105.139, 35.996, -108.502, -0.644, -1604.605]
  MoveL 882 to (57.35, 240.79, 70) mm, rotated rx -90 ry -25 rz 130.88 deg; joints [-4.834, -49.309, 104.898, 36.219, -108.512, -0.911, -1610.878]
  MoveL 883 to (58.51, 247.24, 80) mm, rotated rx -90 ry -25 rz 137.3 deg; joints [-4.463, -49.207, 104.652, 36.44, -108.52, -1.18, -1617.303]
  MoveL 884 to (58.95, 253.96, 90) mm, rotated rx -90 ry -25 rz 143.84 deg; joints [-4.093, -49.103, 104.398, 36.658, -108.525, -1.451, -1623.84]
  MoveL 885 to (58.6, 260.81, 100) mm, rotated rx -90 ry -25 rz 150.45 deg; joints [-3.725, -48.996, 104.139, 36.874, -108.529, -1.725, -1630.453]
  MoveL 886 to (57.44, 267.68, 110) mm, rotated rx -90 ry -25 rz 157.1 deg; joints [-3.358, -48.885, 103.873, 37.087, -108.532, -2, -1637.105]
  MoveL 887 to (55.46, 274.42, 120) mm, rotated rx -90 ry -25 rz 163.76 deg; joints [-2.992, -48.77, 103.601, 37.298, -108.534, -2.277, -1643.762]
  MoveL 888 to (52.68, 280.9, 130) mm, rotated rx -90 ry -25 rz 170.39 deg; joints [-2.628, -48.65, 103.323, 37.508, -108.536, -2.555, -1650.393]
  MoveL 889 to (49.15, 286.99, 140) mm, rotated rx -90 ry -25 rz 176.97 deg; joints [-2.265, -48.526, 103.038, 37.715, -108.537, -2.834, -1656.967]
  MoveL 890 to (44.94, 292.58, 150) mm, rotated rx -90 ry -25 rz -176.55 deg; joints [-1.904, -48.397, 102.748, 37.92, -108.539, -3.113, -1663.455]
  MoveL 891 to (40.17, 297.58, 160) mm, rotated rx -90 ry -25 rz -170.17 deg; joints [-1.544, -48.262, 102.451, 38.123, -108.54, -3.393, -1669.829]
  MoveL 892 to (34.94, 301.92, 170) mm, rotated rx -90 ry -25 rz -163.94 deg; joints [-1.185, -48.122, 102.148, 38.324, -108.543, -3.673, -1676.061]
  MoveL 893 to (29.38, 305.54, 180) mm, rotated rx -90 ry -25 rz -157.88 deg; joints [-0.828, -47.975, 101.839, 38.524, -108.546, -3.953, -1682.125]
  MoveL 894 to (23.62, 308.44, 190) mm, rotated rx -90 ry -25 rz -152.01 deg; joints [-0.473, -47.824, 101.524, 38.721, -108.549, -4.234, -1687.993]
  MoveL 895 to (17.8, 310.63, 200) mm, rotated rx -90 ry -25 rz -146.36 deg; joints [-0.119, -47.666, 101.203, 38.916, -108.553, -4.515, -1693.638]
  MoveL 896 to (12.04, 312.14, 210) mm, rotated rx -90 ry -25 rz -140.97 deg; joints [0.233, -47.503, 100.875, 39.11, -108.557, -4.796, -1699.032]
  MoveL 897 to (6.46, 313.03, 220) mm, rotated rx -90 ry -25 rz -135.85 deg; joints [0.584, -47.335, 100.541, 39.301, -108.561, -5.078, -1704.147]
  MoveL 898 to (1.16, 313.37, 230) mm, rotated rx -90 ry -25 rz -131.05 deg; joints [0.933, -47.161, 100.201, 39.491, -108.565, -5.36, -1708.952]
  MoveL 899 to (-3.78, 313.26, 240) mm, rotated rx -90 ry -25 rz -126.58 deg; joints [1.28, -46.983, 99.855, 39.678, -108.569, -5.643, -1713.419]
  MoveL 900 to (-8.28, 312.8, 250) mm, rotated rx -90 ry -25 rz -122.48 deg; joints [1.626, -46.801, 99.502, 39.863, -108.572, -5.928, -1717.515]
  MoveL 901 to (-12.3, 312.09, 260) mm, rotated rx -90 ry -25 rz -118.79 deg; joints [1.97, -46.614, 99.142, 40.045, -108.574, -6.214, -1721.209]
  MoveL 902 to (-15.8, 311.23, 270) mm, rotated rx -90 ry -25 rz -115.53 deg; joints [2.312, -46.424, 98.777, 40.225, -108.574, -6.502, -1724.467]
  MoveL 903 to (-18.74, 310.33, 280) mm, rotated rx -90 ry -25 rz -112.74 deg; joints [2.653, -46.23, 98.404, 40.402, -108.573, -6.791, -1727.257]
  MoveL 904 to (-21.11, 309.47, 290) mm, rotated rx -90 ry -25 rz -110.46 deg; joints [2.992, -46.033, 98.025, 40.576, -108.57, -7.083, -1729.544]
  Set speed (1000.0 mm/s)
  MoveL 905 to (-21.11, 309.47, 290) mm, rotated rx -90 ry -25 rz -110.46 deg; joints [2.992, -46.033, 98.025, 40.576, -108.57, -7.083, -1729.544]
  Set speed (1000.0 mm/s)
  MoveL 906 to (-34.79, 325.15, 290) mm, rotated rx -90 ry -25 rz -105.16 deg; joints [2.992, -46.913, 97.922, 40.367, -107.822, -7.755, -1734.84]
  MoveL 907 to (-34.79, 325.15, 290) mm, rotated rx -90 ry -25 rz -105.16 deg; joints [2.992, -46.913, 97.922, 40.367, -107.822, -7.755, -1734.84]
  Set speed (60.0 mm/s)
  MoveL 908 to (-31.73, 326.57, 280) mm, rotated rx -90 ry -25 rz -107.49 deg; joints [2.653, -47.114, 98.301, 40.192, -107.82, -7.463, -1732.51]
  MoveL 909 to (-27.92, 328.13, 270) mm, rotated rx -90 ry -25 rz -110.33 deg; joints [2.312, -47.311, 98.673, 40.015, -107.816, -7.174, -1729.668]
  MoveL 910 to (-23.38, 329.69, 260) mm, rotated rx -90 ry -25 rz -113.65 deg; joints [1.97, -47.505, 99.038, 39.835, -107.811, -6.886, -1726.348]
  MoveL 911 to (-18.11, 331.13, 250) mm, rotated rx -90 ry -25 rz -117.42 deg; joints [1.626, -47.696, 99.397, 39.652, -107.803, -6.601, -1722.585]
  MoveL 912 to (-12.17, 332.29, 240) mm, rotated rx -90 ry -25 rz -121.59 deg; joints [1.28, -47.883, 99.75, 39.468, -107.795, -6.317, -1718.413]
  MoveL 913 to (-5.61, 333.04, 230) mm, rotated rx -90 ry -25 rz -126.13 deg; joints [0.933, -48.065, 100.096, 39.281, -107.786, -6.034, -1713.865]
  MoveL 914 to (1.49, 333.22, 220) mm, rotated rx -90 ry -25 rz -131.03 deg; joints [0.584, -48.243, 100.436, 39.091, -107.776, -5.752, -1708.974]
  MoveL 915 to (9.03, 332.72, 210) mm, rotated rx -90 ry -25 rz -136.23 deg; joints [0.233, -48.416, 100.77, 38.9, -107.766, -5.47, -1703.771]
  MoveL 916 to (16.88, 331.41, 200) mm, rotated rx -90 ry -25 rz -141.71 deg; joints [-0.119, -48.583, 101.097, 38.706, -107.756, -5.189, -1698.287]
  MoveL 917 to (24.89, 329.2, 190) mm, rotated rx -90 ry -25 rz -147.45 deg; joints [-0.473, -48.745, 101.419, 38.511, -107.747, -4.908, -1692.553]
  MoveL 918 to (32.91, 326.04, 180) mm, rotated rx -90 ry -25 rz -153.4 deg; joints [-0.828, -48.902, 101.734, 38.314, -107.738, -4.628, -1686.599]
  MoveL 919 to (40.75, 321.89, 170) mm, rotated rx -90 ry -25 rz -159.55 deg; joints [-1.185, -49.052, 102.043, 38.114, -107.729, -4.347, -1680.453]
  MoveL 920 to (48.24, 316.75, 160) mm, rotated rx -90 ry -25 rz -165.85 deg; joints [-1.544, -49.197, 102.347, 37.913, -107.721, -4.067, -1674.145]
  MoveL 921 to (55.2, 310.67, 150) mm, rotated rx -90 ry -25 rz -172.3 deg; joints [-1.904, -49.336, 102.644, 37.71, -107.714, -3.786, -1667.704]
  MoveL 922 to (61.48, 303.74, 140) mm, rotated rx -90 ry -25 rz -178.84 deg; joints [-2.265, -49.47, 102.935, 37.505, -107.707, -3.506, -1661.158]
  MoveL 923 to (66.92, 296.06, 130) mm, rotated rx -90 ry -25 rz 174.54 deg; joints [-2.628, -49.598, 103.22, 37.299, -107.701, -3.226, -1654.539]
  MoveL 924 to (71.41, 287.77, 120) mm, rotated rx -90 ry -25 rz 167.87 deg; joints [-2.992, -49.721, 103.499, 37.09, -107.695, -2.947, -1647.875]
  MoveL 925 to (74.87, 279.04, 110) mm, rotated rx -90 ry -25 rz 161.2 deg; joints [-3.358, -49.84, 103.771, 36.879, -107.688, -2.669, -1641.198]
  MoveL 926 to (77.24, 270.04, 100) mm, rotated rx -90 ry -25 rz 154.54 deg; joints [-3.725, -49.954, 104.038, 36.666, -107.681, -2.392, -1634.542]
  MoveL 927 to (78.53, 260.95, 90) mm, rotated rx -90 ry -25 rz 147.94 deg; joints [-4.093, -50.065, 104.298, 36.451, -107.672, -2.117, -1627.94]
  MoveL 928 to (78.77, 251.96, 80) mm, rotated rx -90 ry -25 rz 141.43 deg; joints [-4.463, -50.172, 104.552, 36.234, -107.663, -1.843, -1621.427]
  MoveL 929 to (78, 243.23, 70) mm, rotated rx -90 ry -25 rz 135.04 deg; joints [-4.834, -50.277, 104.8, 36.014, -107.651, -1.572, -1615.041]
  MoveL 930 to (76.35, 234.91, 60) mm, rotated rx -90 ry -25 rz 128.82 deg; joints [-5.207, -50.379, 105.041, 35.792, -107.637, -1.303, -1608.819]
  MoveL 931 to (73.92, 227.12, 50) mm, rotated rx -90 ry -25 rz 122.8 deg; joints [-5.581, -50.479, 105.276, 35.568, -107.62, -1.036, -1602.802]
  MoveL 932 to (70.87, 219.96, 40) mm, rotated rx -90 ry -25 rz 117.03 deg; joints [-5.956, -50.577, 105.504, 35.341, -107.601, -0.773, -1597.03]
  MoveL 933 to (67.34, 213.5, 30) mm, rotated rx -90 ry -25 rz 111.55 deg; joints [-6.332, -50.674, 105.726, 35.111, -107.579, -0.512, -1591.545]
  MoveL 934 to (63.51, 207.78, 20) mm, rotated rx -90 ry -25 rz 106.39 deg; joints [-6.709, -50.77, 105.941, 34.879, -107.553, -0.254, -1586.389]
  MoveL 935 to (59.54, 202.81, 10) mm, rotated rx -90 ry -25 rz 101.6 deg; joints [-7.088, -50.864, 106.15, 34.645, -107.524, 0, -1581.605]
  MoveL 936 to (55.59, 198.58, 0) mm, rotated rx -90 ry -25 rz 97.23 deg; joints [-7.468, -50.957, 106.353, 34.408, -107.492, 0.252, -1577.234]
  Set speed (1000.0 mm/s)
  MoveL 937 to (55.59, 198.58, 0) mm, rotated rx -90 ry -25 rz 97.23 deg; joints [-7.468, -50.957, 106.353, 34.408, -107.492, 0.252, -1577.234]
  Set speed (1000.0 mm/s)
  MoveL 938 to (-34.79, 325.15, 290) mm, rotated rx -90 ry -25 rz -105.16 deg; joints [2.992, -46.913, 97.922, 40.367, -107.822, -7.755, -1734.84]
  MoveL 939 to (-34.79, 325.15, 290) mm, rotated rx -90 ry -25 rz -105.16 deg; joints [2.992, -46.913, 97.922, 40.367, -107.822, -7.755, -1734.84]
  Set speed (60.0 mm/s)
  MoveL 940 to (-30.72, 304.75, 290) mm, rotated rx -90 ry -25 rz -100.71 deg; joints [2.992, -46.018, 98.027, 40.58, -108.582, -7.072, -1739.294]
  Set speed (1000.0 mm/s)
  MoveL 941 to (-30.72, 304.75, 290) mm, rotated rx -90 ry -25 rz -100.71 deg; joints [2.992, -46.018, 98.027, 40.58, -108.582, -7.072, -1739.294]
  Set speed (1000.0 mm/s)
  MoveL 942 to (55.59, 198.58, 0) mm, rotated rx -90 ry -25 rz 97.23 deg; joints [-7.468, -50.957, 106.353, 34.408, -107.492, 0.252, -1577.234]
  MoveL 943 to (55.59, 198.58, 0) mm, rotated rx -90 ry -25 rz 97.23 deg; joints [-7.468, -50.957, 106.353, 34.408, -107.492, 0.252, -1577.234]
  Set speed (60.0 mm/s)
  MoveL 944 to (45.21, 216.6, 0) mm, rotated rx -90 ry -25 rz 103.54 deg; joints [-7.468, -50.007, 106.445, 34.599, -108.351, 0.872, -1583.543]
  Set speed (1000.0 mm/s)
  MoveL 945 to (45.21, 216.6, 0) mm, rotated rx -90 ry -25 rz 103.54 deg; joints [-7.468, -50.007, 106.445, 34.599, -108.351, 0.872, -1583.543]
  Set speed (1000.0 mm/s)
  MoveL 946 to (55.59, 198.58, 0) mm, rotated rx -90 ry -25 rz 97.23 deg; joints [-7.468, -50.957, 106.353, 34.408, -107.492, 0.252, -1577.234]
  MoveL 947 to (55.59, 198.58, 0) mm, rotated rx -90 ry -25 rz 97.23 deg; joints [-7.468, -50.957, 106.353, 34.408, -107.492, 0.252, -1577.234]
  Set speed (60.0 mm/s)
  MoveL 948 to (59.54, 202.81, 10) mm, rotated rx -90 ry -25 rz 101.6 deg; joints [-7.088, -50.864, 106.15, 34.645, -107.524, 0, -1581.605]
  MoveL 949 to (63.51, 207.78, 20) mm, rotated rx -90 ry -25 rz 106.39 deg; joints [-6.709, -50.77, 105.941, 34.879, -107.553, -0.254, -1586.389]
  MoveL 950 to (67.34, 213.5, 30) mm, rotated rx -90 ry -25 rz 111.55 deg; joints [-6.332, -50.674, 105.726, 35.111, -107.579, -0.512, -1591.545]
  MoveL 951 to (70.87, 219.96, 40) mm, rotated rx -90 ry -25 rz 117.03 deg; joints [-5.956, -50.577, 105.504, 35.341, -107.601, -0.773, -1597.03]
  MoveL 952 to (73.92, 227.12, 50) mm, rotated rx -90 ry -25 rz 122.8 deg; joints [-5.581, -50.479, 105.276, 35.568, -107.62, -1.036, -1602.802]
  MoveL 953 to (76.35, 234.91, 60) mm, rotated rx -90 ry -25 rz 128.82 deg; joints [-5.207, -50.379, 105.041, 35.792, -107.637, -1.303, -1608.819]
  MoveL 954 to (78, 243.23, 70) mm, rotated rx -90 ry -25 rz 135.04 deg; joints [-4.834, -50.277, 104.8, 36.014, -107.651, -1.572, -1615.041]
  MoveL 955 to (78.77, 251.96, 80) mm, rotated rx -90 ry -25 rz 141.43 deg; joints [-4.463, -50.172, 104.552, 36.234, -107.663, -1.843, -1621.427]
  MoveL 956 to (78.53, 260.95, 90) mm, rotated rx -90 ry -25 rz 147.94 deg; joints [-4.093, -50.065, 104.298, 36.451, -107.672, -2.117, -1627.94]
  MoveL 957 to (77.24, 270.04, 100) mm, rotated rx -90 ry -25 rz 154.54 deg; joints [-3.725, -49.954, 104.038, 36.666, -107.681, -2.392, -1634.542]
  MoveL 958 to (74.87, 279.04, 110) mm, rotated rx -90 ry -25 rz 161.2 deg; joints [-3.358, -49.84, 103.771, 36.879, -107.688, -2.669, -1641.198]
  MoveL 959 to (71.41, 287.77, 120) mm, rotated rx -90 ry -25 rz 167.87 deg; joints [-2.992, -49.721, 103.499, 37.09, -107.695, -2.947, -1647.875]
  MoveL 960 to (66.92, 296.06, 130) mm, rotated rx -90 ry -25 rz 174.54 deg; joints [-2.628, -49.598, 103.22, 37.299, -107.701, -3.226, -1654.539]
  MoveL 961 to (61.48, 303.74, 140) mm, rotated rx -90 ry -25 rz -178.84 deg; joints [-2.265, -49.47, 102.935, 37.505, -107.707, -3.506, -1661.158]
  MoveL 962 to (55.2, 310.67, 150) mm, rotated rx -90 ry -25 rz -172.3 deg; joints [-1.904, -49.336, 102.644, 37.71, -107.714, -3.786, -1667.704]
  MoveL 963 to (48.24, 316.75, 160) mm, rotated rx -90 ry -25 rz -165.85 deg; joints [-1.544, -49.197, 102.347, 37.913, -107.721, -4.067, -1674.145]
  MoveL 964 to (40.75, 321.89, 170) mm, rotated rx -90 ry -25 rz -159.55 deg; joints [-1.185, -49.052, 102.043, 38.114, -107.729, -4.347, -1680.453]
  MoveL 965 to (32.91, 326.04, 180) mm, rotated rx -90 ry -25 rz -153.4 deg; joints [-0.828, -48.902, 101.734, 38.314, -107.738, -4.628, -1686.599]
  MoveL 966 to (24.89, 329.2, 190) mm, rotated rx -90 ry -25 rz -147.45 deg; joints [-0.473, -48.745, 101.419, 38.511, -107.747, -4.908, -1692.553]
  MoveL 967 to (16.88, 331.41, 200) mm, rotated rx -90 ry -25 rz -141.71 deg; joints [-0.119, -48.583, 101.097, 38.706, -107.756, -5.189, -1698.287]
  MoveL 968 to (9.03, 332.72, 210) mm, rotated rx -90 ry -25 rz -136.23 deg; joints [0.233, -48.416, 100.77, 38.9, -107.766, -5.47, -1703.771]
  MoveL 969 to (1.49, 333.22, 220) mm, rotated rx -90 ry -25 rz -131.03 deg; joints [0.584, -48.243, 100.436, 39.091, -107.776, -5.752, -1708.974]
  MoveL 970 to (-5.61, 333.04, 230) mm, rotated rx -90 ry -25 rz -126.13 deg; joints [0.933, -48.065, 100.096, 39.281, -107.786, -6.034, -1713.865]
  MoveL 971 to (-12.17, 332.29, 240) mm, rotated rx -90 ry -25 rz -121.59 deg; joints [1.28, -47.883, 99.75, 39.468, -107.795, -6.317, -1718.413]
  MoveL 972 to (-18.11, 331.13, 250) mm, rotated rx -90 ry -25 rz -117.42 deg; joints [1.626, -47.696, 99.397, 39.652, -107.803, -6.601, -1722.585]
  MoveL 973 to (-23.38, 329.69, 260) mm, rotated rx -90 ry -25 rz -113.65 deg; joints [1.97, -47.505, 99.038, 39.835, -107.811, -6.886, -1726.348]
  MoveL 974 to (-27.92, 328.13, 270) mm, rotated rx -90 ry -25 rz -110.33 deg; joints [2.312, -47.311, 98.673, 40.015, -107.816, -7.174, -1729.668]
  MoveL 975 to (-31.73, 326.57, 280) mm, rotated rx -90 ry -25 rz -107.49 deg; joints [2.653, -47.114, 98.301, 40.192, -107.82, -7.463, -1732.51]
  MoveL 976 to (-34.79, 325.15, 290) mm, rotated rx -90 ry -25 rz -105.16 deg; joints [2.992, -46.913, 97.922, 40.367, -107.822, -7.755, -1734.84]
  Set speed (1000.0 mm/s)
  MoveL 977 to (-34.79, 325.15, 290) mm, rotated rx -90 ry -25 rz -105.16 deg; joints [2.992, -46.913, 97.922, 40.367, -107.822, -7.755, -1734.84]
  Set speed (1000.0 mm/s)
  MoveL 978 to (-30.72, 304.75, 290) mm, rotated rx -90 ry -25 rz -100.71 deg; joints [2.992, -46.018, 98.027, 40.58, -108.582, -7.072, -1739.294]
  MoveL 979 to (-30.72, 304.75, 290) mm, rotated rx -90 ry -25 rz -100.71 deg; joints [2.992, -46.018, 98.027, 40.58, -108.582, -7.072, -1739.294]
  Set speed (60.0 mm/s)
  MoveL 980 to (-28.54, 306.02, 280) mm, rotated rx -90 ry -25 rz -103 deg; joints [2.653, -46.216, 98.406, 40.405, -108.584, -6.781, -1736.997]
  MoveL 981 to (-25.81, 307.44, 270) mm, rotated rx -90 ry -25 rz -105.8 deg; joints [2.312, -46.412, 98.778, 40.228, -108.584, -6.493, -1734.195]
  MoveL 982 to (-22.53, 308.91, 260) mm, rotated rx -90 ry -25 rz -109.08 deg; joints [1.97, -46.604, 99.143, 40.047, -108.582, -6.206, -1730.925]
  MoveL 983 to (-18.7, 310.34, 250) mm, rotated rx -90 ry -25 rz -112.78 deg; joints [1.626, -46.793, 99.502, 39.864, -108.579, -5.922, -1727.22]
  MoveL 984 to (-14.35, 311.61, 240) mm, rotated rx -90 ry -25 rz -116.88 deg; joints [1.28, -46.978, 99.855, 39.679, -108.574, -5.639, -1723.116]
  MoveL 985 to (-9.52, 312.61, 230) mm, rotated rx -90 ry -25 rz -121.36 deg; joints [0.933, -47.159, 100.201, 39.491, -108.568, -5.358, -1718.643]
  MoveL 986 to (-4.24, 313.23, 220) mm, rotated rx -90 ry -25 rz -126.16 deg; joints [0.584, -47.335, 100.541, 39.301, -108.561, -5.078, -1713.836]
  MoveL 987 to (1.41, 313.37, 210) mm, rotated rx -90 ry -25 rz -131.27 deg; joints [0.233, -47.507, 100.875, 39.109, -108.554, -4.799, -1708.726]
  MoveL 988 to (7.35, 312.92, 200) mm, rotated rx -90 ry -25 rz -136.66 deg; joints [-0.119, -47.673, 101.202, 38.915, -108.547, -4.52, -1703.341]
  MoveL 989 to (13.47, 311.83, 190) mm, rotated rx -90 ry -25 rz -142.29 deg; joints [-0.473, -47.835, 101.523, 38.718, -108.54, -4.242, -1697.713]
  MoveL 990 to (19.65, 310.01, 180) mm, rotated rx -90 ry -25 rz -148.13 deg; joints [-0.828, -47.99, 101.838, 38.52, -108.533, -3.964, -1691.868]
  MoveL 991 to (25.78, 307.45, 170) mm, rotated rx -90 ry -25 rz -154.16 deg; joints [-1.185, -48.14, 102.146, 38.32, -108.527, -3.686, -1685.836]
  MoveL 992 to (31.7, 304.13, 160) mm, rotated rx -90 ry -25 rz -160.36 deg; joints [-1.544, -48.284, 102.449, 38.118, -108.522, -3.409, -1679.644]
  MoveL 993 to (37.3, 300.08, 150) mm, rotated rx -90 ry -25 rz -166.68 deg; joints [-1.904, -48.422, 102.745, 37.914, -108.517, -3.131, -1673.318]
  MoveL 994 to (42.45, 295.34, 140) mm, rotated rx -90 ry -25 rz -173.11 deg; joints [-2.265, -48.554, 103.036, 37.708, -108.513, -2.854, -1666.886]
  MoveL 995 to (47.02, 289.99, 130) mm, rotated rx -90 ry -25 rz -179.62 deg; joints [-2.628, -48.681, 103.32, 37.501, -108.509, -2.577, -1660.375]
  MoveL 996 to (50.93, 284.12, 120) mm, rotated rx -90 ry -25 rz 173.82 deg; joints [-2.992, -48.803, 103.598, 37.291, -108.505, -2.3, -1653.815]
  MoveL 997 to (54.1, 277.85, 110) mm, rotated rx -90 ry -25 rz 167.23 deg; joints [-3.358, -48.92, 103.87, 37.079, -108.501, -2.025, -1647.235]
  MoveL 998 to (56.49, 271.3, 100) mm, rotated rx -90 ry -25 rz 160.66 deg; joints [-3.725, -49.033, 104.136, 36.866, -108.497, -1.75, -1640.664]
  MoveL 999 to (58.06, 264.62, 90) mm, rotated rx -90 ry -25 rz 154.14 deg; joints [-4.093, -49.141, 104.395, 36.65, -108.492, -1.477, -1634.137]
  MoveL 1000 to (58.85, 257.94, 80) mm, rotated rx -90 ry -25 rz 147.69 deg; joints [-4.463, -49.246, 104.648, 36.431, -108.486, -1.206, -1627.686]
  MoveL 1001 to (58.87, 251.39, 70) mm, rotated rx -90 ry -25 rz 141.35 deg; joints [-4.834, -49.348, 104.895, 36.211, -108.478, -0.937, -1621.348]
  MoveL 1002 to (58.2, 245.07, 60) mm, rotated rx -90 ry -25 rz 135.16 deg; joints [-5.207, -49.447, 105.136, 35.988, -108.468, -0.67, -1615.162]
  MoveL 1003 to (56.92, 239.11, 50) mm, rotated rx -90 ry -25 rz 129.17 deg; joints [-5.581, -49.545, 105.37, 35.763, -108.456, -0.406, -1609.166]
  MoveL 1004 to (55.13, 233.57, 40) mm, rotated rx -90 ry -25 rz 123.4 deg; joints [-5.956, -49.64, 105.598, 35.535, -108.441, -0.144, -1603.403]
  MoveL 1005 to (52.95, 228.52, 30) mm, rotated rx -90 ry -25 rz 117.91 deg; joints [-6.332, -49.733, 105.819, 35.305, -108.423, 0.115, -1597.915]
  MoveL 1006 to (50.48, 223.99, 20) mm, rotated rx -90 ry -25 rz 112.75 deg; joints [-6.709, -49.826, 106.034, 35.072, -108.402, 0.37, -1592.746]
  MoveL 1007 to (47.86, 220.02, 10) mm, rotated rx -90 ry -25 rz 107.94 deg; joints [-7.088, -49.917, 106.243, 34.837, -108.378, 0.623, -1587.94]
  MoveL 1008 to (45.21, 216.6, 0) mm, rotated rx -90 ry -25 rz 103.54 deg; joints [-7.468, -50.007, 106.445, 34.599, -108.351, 0.872, -1583.543]
  Set speed (1000.0 mm/s)
  MoveL 1009 to (45.21, 216.6, 0) mm, rotated rx -90 ry -25 rz 103.54 deg; joints [-7.468, -50.007, 106.445, 34.599, -108.351, 0.872, -1583.543]
  Set speed (1000.0 mm/s)
  MoveL 1010 to (-30.72, 304.75, 290) mm, rotated rx -90 ry -25 rz -100.71 deg; joints [2.992, -46.018, 98.027, 40.58, -108.582, -7.072, -1739.294]
  MoveL 1011 to (-30.72, 304.75, 290) mm, rotated rx -90 ry -25 rz -100.71 deg; joints [2.992, -46.018, 98.027, 40.58, -108.582, -7.072, -1739.294]
  Set speed (60.0 mm/s)
  MoveL 1012 to (-58.22, 263.67, 290) mm, rotated rx -90 ry -25 rz -53.21 deg; joints [2.992, -45.884, 98.039, 40.612, -108.694, -6.971, -1786.787]
  Set speed (1000.0 mm/s)
  MoveL 1013 to (-58.22, 263.67, 290) mm, rotated rx -90 ry -25 rz -53.21 deg; joints [2.992, -45.884, 98.039, 40.612, -108.694, -6.971, -1786.787]
  Set speed (1000.0 mm/s)
  MoveL 1014 to (45.21, 216.6, 0) mm, rotated rx -90 ry -25 rz 103.54 deg; joints [-7.468, -50.007, 106.445, 34.599, -108.351, 0.872, -1943.543]
  MoveL 1015 to (45.21, 216.6, 0) mm, rotated rx -90 ry -25 rz 103.54 deg; joints [-7.468, -50.007, 106.445, 34.599, -108.351, 0.872, -1943.543]
  Set speed (60.0 mm/s)
  MoveL 1016 to (58.12, 264.32, 0) mm, rotated rx -90 ry -25 rz 153.85 deg; joints [-7.468, -50.186, 106.43, 34.563, -108.191, 0.757, -1993.845]
  Set speed (1000.0 mm/s)
  MoveL 1017 to (58.12, 264.32, 0) mm, rotated rx -90 ry -25 rz 153.85 deg; joints [-7.468, -50.186, 106.43, 34.563, -108.191, 0.757, -1993.845]
  Set speed (1000.0 mm/s)
  MoveL 1018 to (45.21, 216.6, 0) mm, rotated rx -90 ry -25 rz 103.54 deg; joints [-7.468, -50.007, 106.445, 34.599, -108.351, 0.872, -1943.543]
  MoveL 1019 to (45.21, 216.6, 0) mm, rotated rx -90 ry -25 rz 103.54 deg; joints [-7.468, -50.007, 106.445, 34.599, -108.351, 0.872, -1943.543]
  Set speed (60.0 mm/s)
  MoveL 1020 to (47.86, 220.02, 10) mm, rotated rx -90 ry -25 rz 107.94 deg; joints [-7.088, -49.917, 106.243, 34.837, -108.378, 0.623, -1947.94]
  MoveL 1021 to (50.48, 223.99, 20) mm, rotated rx -90 ry -25 rz 112.75 deg; joints [-6.709, -49.826, 106.034, 35.072, -108.402, 0.37, -1952.746]
  MoveL 1022 to (52.95, 228.52, 30) mm, rotated rx -90 ry -25 rz 117.91 deg; joints [-6.332, -49.733, 105.819, 35.305, -108.423, 0.115, -1957.915]
  MoveL 1023 to (55.13, 233.57, 40) mm, rotated rx -90 ry -25 rz 123.4 deg; joints [-5.956, -49.64, 105.598, 35.535, -108.441, -0.144, -1963.403]
  MoveL 1024 to (56.92, 239.11, 50) mm, rotated rx -90 ry -25 rz 129.17 deg; joints [-5.581, -49.545, 105.37, 35.763, -108.456, -0.406, -1969.166]
  MoveL 1025 to (58.2, 245.07, 60) mm, rotated rx -90 ry -25 rz 135.16 deg; joints [-5.207, -49.447, 105.136, 35.988, -108.468, -0.67, -1975.162]
  MoveL 1026 to (58.87, 251.39, 70) mm, rotated rx -90 ry -25 rz 141.35 deg; joints [-4.834, -49.348, 104.895, 36.211, -108.478, -0.937, -1981.348]
  MoveL 1027 to (58.85, 257.94, 80) mm, rotated rx -90 ry -25 rz 147.69 deg; joints [-4.463, -49.246, 104.648, 36.431, -108.486, -1.206, -1987.686]
  MoveL 1028 to (58.06, 264.62, 90) mm, rotated rx -90 ry -25 rz 154.14 deg; joints [-4.093, -49.141, 104.395, 36.65, -108.492, -1.477, -1994.137]
  MoveL 1029 to (56.49, 271.3, 100) mm, rotated rx -90 ry -25 rz 160.66 deg; joints [-3.725, -49.033, 104.136, 36.866, -108.497, -1.75, -2000.664]
  MoveL 1030 to (54.1, 277.85, 110) mm, rotated rx -90 ry -25 rz 167.23 deg; joints [-3.358, -48.92, 103.87, 37.079, -108.501, -2.025, -2007.235]
  MoveL 1031 to (50.93, 284.12, 120) mm, rotated rx -90 ry -25 rz 173.82 deg; joints [-2.992, -48.803, 103.598, 37.291, -108.505, -2.3, -2013.815]
  MoveL 1032 to (47.02, 289.99, 130) mm, rotated rx -90 ry -25 rz -179.62 deg; joints [-2.628, -48.681, 103.32, 37.501, -108.509, -2.577, -2020.375]
  MoveL 1033 to (42.45, 295.34, 140) mm, rotated rx -90 ry -25 rz -173.11 deg; joints [-2.265, -48.554, 103.036, 37.708, -108.513, -2.854, -2026.886]
  MoveL 1034 to (37.3, 300.08, 150) mm, rotated rx -90 ry -25 rz -166.68 deg; joints [-1.904, -48.422, 102.745, 37.914, -108.517, -3.131, -2033.318]
  MoveL 1035 to (31.7, 304.13, 160) mm, rotated rx -90 ry -25 rz -160.36 deg; joints [-1.544, -48.284, 102.449, 38.118, -108.522, -3.409, -2039.644]
  MoveL 1036 to (25.78, 307.45, 170) mm, rotated rx -90 ry -25 rz -154.16 deg; joints [-1.185, -48.14, 102.146, 38.32, -108.527, -3.686, -2045.836]
  MoveL 1037 to (19.65, 310.01, 180) mm, rotated rx -90 ry -25 rz -148.13 deg; joints [-0.828, -47.99, 101.838, 38.52, -108.533, -3.964, -2051.868]
  MoveL 1038 to (13.47, 311.83, 190) mm, rotated rx -90 ry -25 rz -142.29 deg; joints [-0.473, -47.835, 101.523, 38.718, -108.54, -4.242, -2057.713]
  MoveL 1039 to (7.35, 312.92, 200) mm, rotated rx -90 ry -25 rz -136.66 deg; joints [-0.119, -47.673, 101.202, 38.915, -108.547, -4.52, -2063.341]
  MoveL 1040 to (1.41, 313.37, 210) mm, rotated rx -90 ry -25 rz -131.27 deg; joints [0.233, -47.507, 100.875, 39.109, -108.554, -4.799, -2068.726]
  MoveL 1041 to (-4.24, 313.23, 220) mm, rotated rx -90 ry -25 rz -126.16 deg; joints [0.584, -47.335, 100.541, 39.301, -108.561, -5.078, -2073.836]
  MoveL 1042 to (-9.52, 312.61, 230) mm, rotated rx -90 ry -25 rz -121.36 deg; joints [0.933, -47.159, 100.201, 39.491, -108.568, -5.358, -2078.643]
  MoveL 1043 to (-14.35, 311.61, 240) mm, rotated rx -90 ry -25 rz -116.88 deg; joints [1.28, -46.978, 99.855, 39.679, -108.574, -5.639, -2083.116]
  MoveL 1044 to (-18.7, 310.34, 250) mm, rotated rx -90 ry -25 rz -112.78 deg; joints [1.626, -46.793, 99.502, 39.864, -108.579, -5.922, -2087.22]
  MoveL 1045 to (-22.53, 308.91, 260) mm, rotated rx -90 ry -25 rz -109.08 deg; joints [1.97, -46.604, 99.143, 40.047, -108.582, -6.206, -2090.925]
  MoveL 1046 to (-25.81, 307.44, 270) mm, rotated rx -90 ry -25 rz -105.8 deg; joints [2.312, -46.412, 98.778, 40.228, -108.584, -6.493, -2094.195]
  MoveL 1047 to (-28.54, 306.02, 280) mm, rotated rx -90 ry -25 rz -103 deg; joints [2.653, -46.216, 98.406, 40.405, -108.584, -6.781, -2096.997]
  MoveL 1048 to (-30.72, 304.75, 290) mm, rotated rx -90 ry -25 rz -100.71 deg; joints [2.992, -46.018, 98.027, 40.58, -108.582, -7.072, -2099.294]
  Set speed (1000.0 mm/s)
  MoveL 1049 to (-30.72, 304.75, 290) mm, rotated rx -90 ry -25 rz -100.71 deg; joints [2.992, -46.018, 98.027, 40.58, -108.582, -7.072, -2099.294]
  Set speed (1000.0 mm/s)
  MoveL 1050 to (-58.22, 263.67, 290) mm, rotated rx -90 ry -25 rz -53.21 deg; joints [2.992, -45.884, 98.039, 40.612, -108.694, -6.971, -2146.787]
  MoveL 1051 to (-58.22, 263.67, 290) mm, rotated rx -90 ry -25 rz -53.21 deg; joints [2.992, -45.884, 98.039, 40.612, -108.694, -6.971, -2146.787]
  Set speed (60.0 mm/s)
  MoveL 1052 to (-57.77, 266.15, 280) mm, rotated rx -90 ry -25 rz -55.62 deg; joints [2.653, -46.086, 98.418, 40.436, -108.693, -6.683, -2144.382]
  MoveL 1053 to (-57.08, 269.15, 270) mm, rotated rx -90 ry -25 rz -58.54 deg; joints [2.312, -46.286, 98.79, 40.257, -108.689, -6.399, -2141.455]
  MoveL 1054 to (-56.08, 272.6, 260) mm, rotated rx -90 ry -25 rz -61.95 deg; joints [1.97, -46.485, 99.155, 40.076, -108.682, -6.118, -2138.047]
  MoveL 1055 to (-54.69, 276.44, 250) mm, rotated rx -90 ry -25 rz -65.8 deg; joints [1.626, -46.682, 99.513, 39.891, -108.672, -5.84, -2134.197]
  MoveL 1056 to (-52.84, 280.57, 240) mm, rotated rx -90 ry -25 rz -70.06 deg; joints [1.28, -46.876, 99.865, 39.703, -108.659, -5.564, -2129.944]
  MoveL 1057 to (-50.46, 284.91, 230) mm, rotated rx -90 ry -25 rz -74.67 deg; joints [0.933, -47.068, 100.21, 39.513, -108.644, -5.292, -2125.328]
  MoveL 1058 to (-47.51, 289.33, 220) mm, rotated rx -90 ry -25 rz -79.61 deg; joints [0.584, -47.257, 100.549, 39.32, -108.627, -5.021, -2120.386]
  MoveL 1059 to (-43.95, 293.72, 210) mm, rotated rx -90 ry -25 rz -84.84 deg; joints [0.233, -47.443, 100.881, 39.124, -108.608, -4.752, -2115.156]
  MoveL 1060 to (-39.77, 297.95, 200) mm, rotated rx -90 ry -25 rz -90.33 deg; joints [-0.119, -47.624, 101.206, 38.926, -108.588, -4.485, -2109.672]
  MoveL 1061 to (-34.96, 301.9, 190) mm, rotated rx -90 ry -25 rz -96.03 deg; joints [-0.473, -47.802, 101.526, 38.726, -108.567, -4.218, -2103.97]
  MoveL 1062 to (-29.57, 305.43, 180) mm, rotated rx -90 ry -25 rz -101.92 deg; joints [-0.828, -47.975, 101.839, 38.524, -108.546, -3.953, -2098.081]
  MoveL 1063 to (-23.65, 308.43, 170) mm, rotated rx -90 ry -25 rz -107.96 deg; joints [-1.185, -48.143, 102.146, 38.319, -108.524, -3.689, -2092.038]
  MoveL 1064 to (-17.28, 310.79, 160) mm, rotated rx -90 ry -25 rz -114.13 deg; joints [-1.544, -48.306, 102.447, 38.113, -108.503, -3.424, -2085.87]
  MoveL 1065 to (-10.57, 312.43, 150) mm, rotated rx -90 ry -25 rz -120.39 deg; joints [-1.904, -48.463, 102.742, 37.905, -108.481, -3.16, -2079.606]
  MoveL 1066 to (-3.62, 313.27, 140) mm, rotated rx -90 ry -25 rz -126.72 deg; joints [-2.265, -48.614, 103.03, 37.695, -108.461, -2.896, -2073.276]
  MoveL 1067 to (3.42, 313.28, 130) mm, rotated rx -90 ry -25 rz -133.09 deg; joints [-2.628, -48.76, 103.313, 37.483, -108.441, -2.632, -2066.906]
  MoveL 1068 to (10.42, 312.45, 120) mm, rotated rx -90 ry -25 rz -139.47 deg; joints [-2.992, -48.899, 103.589, 37.27, -108.422, -2.367, -2060.525]
  MoveL 1069 to (17.25, 310.8, 110) mm, rotated rx -90 ry -25 rz -145.84 deg; joints [-3.358, -49.032, 103.86, 37.055, -108.404, -2.103, -2054.159]
  MoveL 1070 to (23.78, 308.38, 100) mm, rotated rx -90 ry -25 rz -152.16 deg; joints [-3.725, -49.16, 104.124, 36.838, -108.386, -1.838, -2047.838]
  MoveL 1071 to (29.89, 305.25, 90) mm, rotated rx -90 ry -25 rz -158.41 deg; joints [-4.093, -49.282, 104.382, 36.619, -108.369, -1.574, -2041.588]
  MoveL 1072 to (35.48, 301.51, 80) mm, rotated rx -90 ry -25 rz -164.56 deg; joints [-4.463, -49.398, 104.635, 36.399, -108.352, -1.31, -2035.44]
  MoveL 1073 to (40.49, 297.28, 70) mm, rotated rx -90 ry -25 rz -170.58 deg; joints [-4.834, -49.51, 104.881, 36.176, -108.336, -1.047, -2029.423]
  MoveL 1074 to (44.86, 292.68, 60) mm, rotated rx -90 ry -25 rz -176.43 deg; joints [-5.207, -49.617, 105.121, 35.952, -108.319, -0.784, -2023.57]
  MoveL 1075 to (48.58, 287.83, 50) mm, rotated rx -90 ry -25 rz 177.91 deg; joints [-5.581, -49.72, 105.355, 35.726, -108.302, -0.523, -2017.914]
  MoveL 1076 to (51.63, 282.88, 40) mm, rotated rx -90 ry -25 rz 172.49 deg; joints [-5.956, -49.819, 105.582, 35.498, -108.283, -0.263, -2012.49]
  MoveL 1077 to (54.06, 277.94, 30) mm, rotated rx -90 ry -25 rz 167.33 deg; joints [-6.332, -49.914, 105.804, 35.267, -108.263, -0.005, -2007.332]
  MoveL 1078 to (55.91, 273.13, 20) mm, rotated rx -90 ry -25 rz 162.48 deg; joints [-6.709, -50.007, 106.019, 35.035, -108.241, 0.251, -2002.48]
  MoveL 1079 to (57.23, 268.56, 10) mm, rotated rx -90 ry -25 rz 157.97 deg; joints [-7.088, -50.097, 106.227, 34.8, -108.218, 0.505, -1997.971]
  MoveL 1080 to (58.12, 264.32, 0) mm, rotated rx -90 ry -25 rz 153.85 deg; joints [-7.468, -50.186, 106.43, 34.563, -108.191, 0.757, -1993.845]
  Set speed (1000.0 mm/s)
  MoveL 1081 to (58.12, 264.32, 0) mm, rotated rx -90 ry -25 rz 153.85 deg; joints [-7.468, -50.186, 106.43, 34.563, -108.191, 0.757, -1993.845]
  Set speed (1000.0 mm/s)
  MoveL 1082 to (-58.22, 263.67, 290) mm, rotated rx -90 ry -25 rz -53.21 deg; joints [2.992, -45.884, 98.039, 40.612, -108.694, -6.971, -2146.787]
  MoveL 1083 to (-58.22, 263.67, 290) mm, rotated rx -90 ry -25 rz -53.21 deg; joints [2.992, -45.884, 98.039, 40.612, -108.694, -6.971, -2146.787]
  Set speed (60.0 mm/s)
  MoveL 1084 to (-78.63, 259.66, 290) mm, rotated rx -90 ry -25 rz -47.01 deg; joints [2.992, -46.754, 97.943, 40.404, -107.959, -7.632, -2152.994]
  Set speed (1000.0 mm/s)
  MoveL 1085 to (-78.63, 259.66, 290) mm, rotated rx -90 ry -25 rz -47.01 deg; joints [2.992, -46.754, 97.943, 40.404, -107.959, -7.632, -2152.994]
  Set speed (1000.0 mm/s)
  MoveL 1086 to (58.12, 264.32, 0) mm, rotated rx -90 ry -25 rz 153.85 deg; joints [-7.468, -50.186, 106.43, 34.563, -108.191, 0.757, -1993.845]
  MoveL 1087 to (58.12, 264.32, 0) mm, rotated rx -90 ry -25 rz 153.85 deg; joints [-7.468, -50.186, 106.43, 34.563, -108.191, 0.757, -1993.845]
  Set speed (60.0 mm/s)
  MoveL 1088 to (76.17, 274.65, 0) mm, rotated rx -90 ry -25 rz 157.93 deg; joints [-7.468, -51.166, 106.328, 34.367, -107.299, 0.114, -1997.935]
  Set speed (1000.0 mm/s)
  MoveL 1089 to (76.17, 274.65, 0) mm, rotated rx -90 ry -25 rz 157.93 deg; joints [-7.468, -51.166, 106.328, 34.367, -107.299, 0.114, -1997.935]
  Set speed (1000.0 mm/s)
  MoveL 1090 to (58.12, 264.32, 0) mm, rotated rx -90 ry -25 rz 153.85 deg; joints [-7.468, -50.186, 106.43, 34.563, -108.191, 0.757, -1993.845]
  MoveL 1091 to (58.12, 264.32, 0) mm, rotated rx -90 ry -25 rz 153.85 deg; joints [-7.468, -50.186, 106.43, 34.563, -108.191, 0.757, -1993.845]
  Set speed (60.0 mm/s)
  MoveL 1092 to (57.23, 268.56, 10) mm, rotated rx -90 ry -25 rz 157.97 deg; joints [-7.088, -50.097, 106.227, 34.8, -108.218, 0.505, -1997.971]
  MoveL 1093 to (55.91, 273.13, 20) mm, rotated rx -90 ry -25 rz 162.48 deg; joints [-6.709, -50.007, 106.019, 35.035, -108.241, 0.251, -2002.48]
  MoveL 1094 to (54.06, 277.94, 30) mm, rotated rx -90 ry -25 rz 167.33 deg; joints [-6.332, -49.914, 105.804, 35.267, -108.263, -0.005, -2007.332]
  MoveL 1095 to (51.63, 282.88, 40) mm, rotated rx -90 ry -25 rz 172.49 deg; joints [-5.956, -49.819, 105.582, 35.498, -108.283, -0.263, -2012.49]
  MoveL 1096 to (48.58, 287.83, 50) mm, rotated rx -90 ry -25 rz 177.91 deg; joints [-5.581, -49.72, 105.355, 35.726, -108.302, -0.523, -2017.914]
  MoveL 1097 to (44.86, 292.68, 60) mm, rotated rx -90 ry -25 rz -176.43 deg; joints [-5.207, -49.617, 105.121, 35.952, -108.319, -0.784, -2023.57]
  MoveL 1098 to (40.49, 297.28, 70) mm, rotated rx -90 ry -25 rz -170.58 deg; joints [-4.834, -49.51, 104.881, 36.176, -108.336, -1.047, -2029.423]
  MoveL 1099 to (35.48, 301.51, 80) mm, rotated rx -90 ry -25 rz -164.56 deg; joints [-4.463, -49.398, 104.635, 36.399, -108.352, -1.31, -2035.44]
  MoveL 1100 to (29.89, 305.25, 90) mm, rotated rx -90 ry -25 rz -158.41 deg; joints [-4.093, -49.282, 104.382, 36.619, -108.369, -1.574, -2041.588]
  MoveL 1101 to (23.78, 308.38, 100) mm, rotated rx -90 ry -25 rz -152.16 deg; joints [-3.725, -49.16, 104.124, 36.838, -108.386, -1.838, -2047.838]
  MoveL 1102 to (17.25, 310.8, 110) mm, rotated rx -90 ry -25 rz -145.84 deg; joints [-3.358, -49.032, 103.86, 37.055, -108.404, -2.103, -2054.159]
  MoveL 1103 to (10.42, 312.45, 120) mm, rotated rx -90 ry -25 rz -139.47 deg; joints [-2.992, -48.899, 103.589, 37.27, -108.422, -2.367, -2060.525]
  MoveL 1104 to (3.42, 313.28, 130) mm, rotated rx -90 ry -25 rz -133.09 deg; joints [-2.628, -48.76, 103.313, 37.483, -108.441, -2.632, -2066.906]
  MoveL 1105 to (-3.62, 313.27, 140) mm, rotated rx -90 ry -25 rz -126.72 deg; joints [-2.265, -48.614, 103.03, 37.695, -108.461, -2.896, -2073.276]
  MoveL 1106 to (-10.57, 312.43, 150) mm, rotated rx -90 ry -25 rz -120.39 deg; joints [-1.904, -48.463, 102.742, 37.905, -108.481, -3.16, -2079.606]
  MoveL 1107 to (-17.28, 310.79, 160) mm, rotated rx -90 ry -25 rz -114.13 deg; joints [-1.544, -48.306, 102.447, 38.113, -108.503, -3.424, -2085.87]
  MoveL 1108 to (-23.65, 308.43, 170) mm, rotated rx -90 ry -25 rz -107.96 deg; joints [-1.185, -48.143, 102.146, 38.319, -108.524, -3.689, -2092.038]
  MoveL 1109 to (-29.57, 305.43, 180) mm, rotated rx -90 ry -25 rz -101.92 deg; joints [-0.828, -47.975, 101.839, 38.524, -108.546, -3.953, -2098.081]
  MoveL 1110 to (-34.96, 301.9, 190) mm, rotated rx -90 ry -25 rz -96.03 deg; joints [-0.473, -47.802, 101.526, 38.726, -108.567, -4.218, -2103.97]
  MoveL 1111 to (-39.77, 297.95, 200) mm, rotated rx -90 ry -25 rz -90.33 deg; joints [-0.119, -47.624, 101.206, 38.926, -108.588, -4.485, -2109.672]
  MoveL 1112 to (-43.95, 293.72, 210) mm, rotated rx -90 ry -25 rz -84.84 deg; joints [0.233, -47.443, 100.881, 39.124, -108.608, -4.752, -2115.156]
  MoveL 1113 to (-47.51, 289.33, 220) mm, rotated rx -90 ry -25 rz -79.61 deg; joints [0.584, -47.257, 100.549, 39.32, -108.627, -5.021, -2120.386]
  MoveL 1114 to (-50.46, 284.91, 230) mm, rotated rx -90 ry -25 rz -74.67 deg; joints [0.933, -47.068, 100.21, 39.513, -108.644, -5.292, -2125.328]
  MoveL 1115 to (-52.84, 280.57, 240) mm, rotated rx -90 ry -25 rz -70.06 deg; joints [1.28, -46.876, 99.865, 39.703, -108.659, -5.564, -2129.944]
  MoveL 1116 to (-54.69, 276.44, 250) mm, rotated rx -90 ry -25 rz -65.8 deg; joints [1.626, -46.682, 99.513, 39.891, -108.672, -5.84, -2134.197]
  MoveL 1117 to (-56.08, 272.6, 260) mm, rotated rx -90 ry -25 rz -61.95 deg; joints [1.97, -46.485, 99.155, 40.076, -108.682, -6.118, -2138.047]
  MoveL 1118 to (-57.08, 269.15, 270) mm, rotated rx -90 ry -25 rz -58.54 deg; joints [2.312, -46.286, 98.79, 40.257, -108.689, -6.399, -2141.455]
  MoveL 1119 to (-57.77, 266.15, 280) mm, rotated rx -90 ry -25 rz -55.62 deg; joints [2.653, -46.086, 98.418, 40.436, -108.693, -6.683, -2144.382]
  MoveL 1120 to (-58.22, 263.67, 290) mm, rotated rx -90 ry -25 rz -53.21 deg; joints [2.992, -45.884, 98.039, 40.612, -108.694, -6.971, -2146.787]
  Set speed (1000.0 mm/s)
  MoveL 1121 to (-58.22, 263.67, 290) mm, rotated rx -90 ry -25 rz -53.21 deg; joints [2.992, -45.884, 98.039, 40.612, -108.694, -6.971, -2146.787]
  Set speed (1000.0 mm/s)
  MoveL 1122 to (-78.63, 259.66, 290) mm, rotated rx -90 ry -25 rz -47.01 deg; joints [2.992, -46.754, 97.943, 40.404, -107.959, -7.632, -2152.994]
  MoveL 1123 to (-78.63, 259.66, 290) mm, rotated rx -90 ry -25 rz -47.01 deg; joints [2.992, -46.754, 97.943, 40.404, -107.959, -7.632, -2152.994]
  Set speed (60.0 mm/s)
  MoveL 1124 to (-78.34, 263.02, 280) mm, rotated rx -90 ry -25 rz -49.44 deg; joints [2.653, -46.959, 98.321, 40.229, -107.954, -7.345, -2150.563]
  MoveL 1125 to (-77.78, 267.1, 270) mm, rotated rx -90 ry -25 rz -52.4 deg; joints [2.312, -47.163, 98.693, 40.05, -107.945, -7.06, -2147.603]
  MoveL 1126 to (-76.86, 271.82, 260) mm, rotated rx -90 ry -25 rz -55.85 deg; joints [1.97, -47.365, 99.057, 39.868, -107.933, -6.779, -2144.153]
  MoveL 1127 to (-75.48, 277.1, 250) mm, rotated rx -90 ry -25 rz -59.75 deg; joints [1.626, -47.564, 99.415, 39.683, -107.918, -6.501, -2140.252]
  MoveL 1128 to (-73.51, 282.82, 240) mm, rotated rx -90 ry -25 rz -64.06 deg; joints [1.28, -47.762, 99.766, 39.496, -107.901, -6.225, -2135.94]
  MoveL 1129 to (-70.88, 288.88, 230) mm, rotated rx -90 ry -25 rz -68.74 deg; joints [0.933, -47.957, 100.111, 39.305, -107.88, -5.952, -2131.255]
  MoveL 1130 to (-67.49, 295.12, 220) mm, rotated rx -90 ry -25 rz -73.76 deg; joints [0.584, -48.15, 100.449, 39.113, -107.858, -5.682, -2126.236]
  MoveL 1131 to (-63.28, 301.4, 210) mm, rotated rx -90 ry -25 rz -79.08 deg; joints [0.233, -48.339, 100.78, 38.917, -107.834, -5.413, -2120.918]
  MoveL 1132 to (-58.22, 307.54, 200) mm, rotated rx -90 ry -25 rz -84.66 deg; joints [-0.119, -48.525, 101.105, 38.72, -107.808, -5.146, -2115.34]
  MoveL 1133 to (-52.31, 313.38, 190) mm, rotated rx -90 ry -25 rz -90.47 deg; joints [-0.473, -48.707, 101.424, 38.52, -107.781, -4.88, -2109.535]
  MoveL 1134 to (-45.56, 318.73, 180) mm, rotated rx -90 ry -25 rz -96.46 deg; joints [-0.828, -48.884, 101.737, 38.318, -107.754, -4.615, -2103.538]
  MoveL 1135 to (-38.04, 323.45, 170) mm, rotated rx -90 ry -25 rz -102.62 deg; joints [-1.185, -49.056, 102.043, 38.113, -107.726, -4.35, -2097.381]
  MoveL 1136 to (-29.85, 327.37, 160) mm, rotated rx -90 ry -25 rz -108.9 deg; joints [-1.544, -49.223, 102.343, 37.907, -107.698, -4.086, -2091.097]
  MoveL 1137 to (-21.11, 330.36, 150) mm, rotated rx -90 ry -25 rz -115.28 deg; joints [-1.904, -49.385, 102.637, 37.7, -107.67, -3.822, -2084.715]
  MoveL 1138 to (-11.96, 332.32, 140) mm, rotated rx -90 ry -25 rz -121.73 deg; joints [-2.265, -49.541, 102.926, 37.49, -107.643, -3.558, -2078.268]
  MoveL 1139 to (-2.59, 333.2, 130) mm, rotated rx -90 ry -25 rz -128.22 deg; joints [-2.628, -49.691, 103.208, 37.278, -107.617, -3.293, -2071.782]
  MoveL 1140 to (6.83, 332.94, 120) mm, rotated rx -90 ry -25 rz -134.71 deg; joints [-2.992, -49.835, 103.484, 37.065, -107.592, -3.029, -2065.289]
  MoveL 1141 to (16.13, 331.57, 110) mm, rotated rx -90 ry -25 rz -141.18 deg; joints [-3.358, -49.973, 103.754, 36.851, -107.568, -2.764, -2058.817]
  MoveL 1142 to (25.11, 329.13, 100) mm, rotated rx -90 ry -25 rz -147.6 deg; joints [-3.725, -50.105, 104.019, 36.634, -107.544, -2.499, -2052.396]
  MoveL 1143 to (33.62, 325.71, 90) mm, rotated rx -90 ry -25 rz -153.95 deg; joints [-4.093, -50.231, 104.277, 36.416, -107.521, -2.234, -2046.054]
  MoveL 1144 to (41.52, 321.41, 80) mm, rotated rx -90 ry -25 rz -160.18 deg; joints [-4.463, -50.352, 104.53, 36.196, -107.499, -1.969, -2039.824]
  MoveL 1145 to (48.7, 316.39, 70) mm, rotated rx -90 ry -25 rz -166.26 deg; joints [-4.834, -50.468, 104.776, 35.974, -107.477, -1.704, -2033.735]
  MoveL 1146 to (55.08, 310.79, 60) mm, rotated rx -90 ry -25 rz -172.18 deg; joints [-5.207, -50.578, 105.016, 35.751, -107.455, -1.44, -2027.821]
  MoveL 1147 to (60.61, 304.79, 50) mm, rotated rx -90 ry -25 rz -177.89 deg; joints [-5.581, -50.685, 105.251, 35.525, -107.432, -1.177, -2022.113]
  MoveL 1148 to (65.29, 298.57, 40) mm, rotated rx -90 ry -25 rz 176.65 deg; joints [-5.956, -50.787, 105.479, 35.298, -107.409, -0.915, -2016.648]
  MoveL 1149 to (69.12, 292.29, 30) mm, rotated rx -90 ry -25 rz 171.46 deg; joints [-6.332, -50.886, 105.701, 35.068, -107.384, -0.655, -2011.461]
  MoveL 1150 to (72.16, 286.11, 20) mm, rotated rx -90 ry -25 rz 166.59 deg; joints [-6.709, -50.982, 105.916, 34.837, -107.358, -0.397, -2006.587]
  MoveL 1151 to (74.48, 280.19, 10) mm, rotated rx -90 ry -25 rz 162.07 deg; joints [-7.088, -51.075, 106.125, 34.603, -107.33, -0.14, -2002.066]
  MoveL 1152 to (76.17, 274.65, 0) mm, rotated rx -90 ry -25 rz 157.93 deg; joints [-7.468, -51.166, 106.328, 34.367, -107.299, 0.114, -1997.935]
  Set speed (1000.0 mm/s)
  MoveL 1153 to (76.17, 274.65, 0) mm, rotated rx -90 ry -25 rz 157.93 deg; joints [-7.468, -51.166, 106.328, 34.367, -107.299, 0.114, -1997.935]
  Set speed (1000.0 mm/s)
  MoveL 1154 to (-78.63, 259.66, 290) mm, rotated rx -90 ry -25 rz -47.01 deg; joints [2.992, -46.754, 97.943, 40.404, -107.959, -7.632, -2152.994]
  MoveL 1155 to (-78.63, 259.66, 290) mm, rotated rx -90 ry -25 rz -47.01 deg; joints [2.992, -46.754, 97.943, 40.404, -107.959, -7.632, -2152.994]
  Set speed (60.0 mm/s)
  MoveL 1156 to (-58.93, 252.99, 290) mm, rotated rx -90 ry -25 rz -42.9 deg; joints [2.992, -45.848, 98.043, 40.621, -108.724, -6.944, -2157.096]
  Set speed (1000.0 mm/s)
  MoveL 1157 to (-58.93, 252.99, 290) mm, rotated rx -90 ry -25 rz -42.9 deg; joints [2.992, -45.848, 98.043, 40.621, -108.724, -6.944, -2157.096]
  Set speed (1000.0 mm/s)
  MoveL 1158 to (76.17, 274.65, 0) mm, rotated rx -90 ry -25 rz 157.93 deg; joints [-7.468, -51.166, 106.328, 34.367, -107.299, 0.114, -1997.935]
  MoveL 1159 to (76.17, 274.65, 0) mm, rotated rx -90 ry -25 rz 157.93 deg; joints [-7.468, -51.166, 106.328, 34.367, -107.299, 0.114, -1997.935]
  Set speed (60.0 mm/s)
  MoveL 1160 to (55.37, 274.67, 0) mm, rotated rx -90 ry -25 rz 164.01 deg; joints [-7.468, -50.223, 106.427, 34.556, -108.158, 0.732, -2004.014]
  Set speed (1000.0 mm/s)
  MoveL 1161 to (55.37, 274.67, 0) mm, rotated rx -90 ry -25 rz 164.01 deg; joints [-7.468, -50.223, 106.427, 34.556, -108.158, 0.732, -2004.014]
  Set speed (1000.0 mm/s)
  MoveL 1162 to (76.17, 274.65, 0) mm, rotated rx -90 ry -25 rz 157.93 deg; joints [-7.468, -51.166, 106.328, 34.367, -107.299, 0.114, -1997.935]
  MoveL 1163 to (76.17, 274.65, 0) mm, rotated rx -90 ry -25 rz 157.93 deg; joints [-7.468, -51.166, 106.328, 34.367, -107.299, 0.114, -1997.935]
  Set speed (60.0 mm/s)
  MoveL 1164 to (74.48, 280.19, 10) mm, rotated rx -90 ry -25 rz 162.07 deg; joints [-7.088, -51.075, 106.125, 34.603, -107.33, -0.14, -2002.066]
  MoveL 1165 to (72.16, 286.11, 20) mm, rotated rx -90 ry -25 rz 166.59 deg; joints [-6.709, -50.982, 105.916, 34.837, -107.358, -0.397, -2006.587]
  MoveL 1166 to (69.12, 292.29, 30) mm, rotated rx -90 ry -25 rz 171.46 deg; joints [-6.332, -50.886, 105.701, 35.068, -107.384, -0.655, -2011.461]
  MoveL 1167 to (65.29, 298.57, 40) mm, rotated rx -90 ry -25 rz 176.65 deg; joints [-5.956, -50.787, 105.479, 35.298, -107.409, -0.915, -2016.648]
  MoveL 1168 to (60.61, 304.79, 50) mm, rotated rx -90 ry -25 rz -177.89 deg; joints [-5.581, -50.685, 105.251, 35.525, -107.432, -1.177, -2022.113]
  MoveL 1169 to (55.08, 310.79, 60) mm, rotated rx -90 ry -25 rz -172.18 deg; joints [-5.207, -50.578, 105.016, 35.751, -107.455, -1.44, -2027.821]
  MoveL 1170 to (48.7, 316.39, 70) mm, rotated rx -90 ry -25 rz -166.26 deg; joints [-4.834, -50.468, 104.776, 35.974, -107.477, -1.704, -2033.735]
  MoveL 1171 to (41.52, 321.41, 80) mm, rotated rx -90 ry -25 rz -160.18 deg; joints [-4.463, -50.352, 104.53, 36.196, -107.499, -1.969, -2039.824]
  MoveL 1172 to (33.62, 325.71, 90) mm, rotated rx -90 ry -25 rz -153.95 deg; joints [-4.093, -50.231, 104.277, 36.416, -107.521, -2.234, -2046.054]
  MoveL 1173 to (25.11, 329.13, 100) mm, rotated rx -90 ry -25 rz -147.6 deg; joints [-3.725, -50.105, 104.019, 36.634, -107.544, -2.499, -2052.396]
  MoveL 1174 to (16.13, 331.57, 110) mm, rotated rx -90 ry -25 rz -141.18 deg; joints [-3.358, -49.973, 103.754, 36.851, -107.568, -2.764, -2058.817]
  MoveL 1175 to (6.83, 332.94, 120) mm, rotated rx -90 ry -25 rz -134.71 deg; joints [-2.992, -49.835, 103.484, 37.065, -107.592, -3.029, -2065.289]
  MoveL 1176 to (-2.59, 333.2, 130) mm, rotated rx -90 ry -25 rz -128.22 deg; joints [-2.628, -49.691, 103.208, 37.278, -107.617, -3.293, -2071.782]
  MoveL 1177 to (-11.96, 332.32, 140) mm, rotated rx -90 ry -25 rz -121.73 deg; joints [-2.265, -49.541, 102.926, 37.49, -107.643, -3.558, -2078.268]
  MoveL 1178 to (-21.11, 330.36, 150) mm, rotated rx -90 ry -25 rz -115.28 deg; joints [-1.904, -49.385, 102.637, 37.7, -107.67, -3.822, -2084.715]
  MoveL 1179 to (-29.85, 327.37, 160) mm, rotated rx -90 ry -25 rz -108.9 deg; joints [-1.544, -49.223, 102.343, 37.907, -107.698, -4.086, -2091.097]
  MoveL 1180 to (-38.04, 323.45, 170) mm, rotated rx -90 ry -25 rz -102.62 deg; joints [-1.185, -49.056, 102.043, 38.113, -107.726, -4.35, -2097.381]
  MoveL 1181 to (-45.56, 318.73, 180) mm, rotated rx -90 ry -25 rz -96.46 deg; joints [-0.828, -48.884, 101.737, 38.318, -107.754, -4.615, -2103.538]
  MoveL 1182 to (-52.31, 313.38, 190) mm, rotated rx -90 ry -25 rz -90.47 deg; joints [-0.473, -48.707, 101.424, 38.52, -107.781, -4.88, -2109.535]
  MoveL 1183 to (-58.22, 307.54, 200) mm, rotated rx -90 ry -25 rz -84.66 deg; joints [-0.119, -48.525, 101.105, 38.72, -107.808, -5.146, -2115.34]
  MoveL 1184 to (-63.28, 301.4, 210) mm, rotated rx -90 ry -25 rz -79.08 deg; joints [0.233, -48.339, 100.78, 38.917, -107.834, -5.413, -2120.918]
  MoveL 1185 to (-67.49, 295.12, 220) mm, rotated rx -90 ry -25 rz -73.76 deg; joints [0.584, -48.15, 100.449, 39.113, -107.858, -5.682, -2126.236]
  MoveL 1186 to (-70.88, 288.88, 230) mm, rotated rx -90 ry -25 rz -68.74 deg; joints [0.933, -47.957, 100.111, 39.305, -107.88, -5.952, -2131.255]
  MoveL 1187 to (-73.51, 282.82, 240) mm, rotated rx -90 ry -25 rz -64.06 deg; joints [1.28, -47.762, 99.766, 39.496, -107.901, -6.225, -2135.94]
  MoveL 1188 to (-75.48, 277.1, 250) mm, rotated rx -90 ry -25 rz -59.75 deg; joints [1.626, -47.564, 99.415, 39.683, -107.918, -6.501, -2140.252]
  MoveL 1189 to (-76.86, 271.82, 260) mm, rotated rx -90 ry -25 rz -55.85 deg; joints [1.97, -47.365, 99.057, 39.868, -107.933, -6.779, -2144.153]
  MoveL 1190 to (-77.78, 267.1, 270) mm, rotated rx -90 ry -25 rz -52.4 deg; joints [2.312, -47.163, 98.693, 40.05, -107.945, -7.06, -2147.603]
  MoveL 1191 to (-78.34, 263.02, 280) mm, rotated rx -90 ry -25 rz -49.44 deg; joints [2.653, -46.959, 98.321, 40.229, -107.954, -7.345, -2150.563]
  MoveL 1192 to (-78.63, 259.66, 290) mm, rotated rx -90 ry -25 rz -47.01 deg; joints [2.992, -46.754, 97.943, 40.404, -107.959, -7.632, -2152.994]
  Set speed (1000.0 mm/s)
  MoveL 1193 to (-78.63, 259.66, 290) mm, rotated rx -90 ry -25 rz -47.01 deg; joints [2.992, -46.754, 97.943, 40.404, -107.959, -7.632, -2152.994]
  Set speed (1000.0 mm/s)
  MoveL 1194 to (-58.93, 252.99, 290) mm, rotated rx -90 ry -25 rz -42.9 deg; joints [2.992, -45.848, 98.043, 40.621, -108.724, -6.944, -2157.096]
  MoveL 1195 to (-58.93, 252.99, 290) mm, rotated rx -90 ry -25 rz -42.9 deg; joints [2.992, -45.848, 98.043, 40.621, -108.724, -6.944, -2157.096]
  Set speed (60.0 mm/s)
  MoveL 1196 to (-58.94, 255.51, 280) mm, rotated rx -90 ry -25 rz -45.34 deg; joints [2.653, -46.05, 98.421, 40.445, -108.723, -6.656, -2154.659]
  MoveL 1197 to (-58.8, 258.59, 270) mm, rotated rx -90 ry -25 rz -48.31 deg; joints [2.312, -46.251, 98.793, 40.266, -108.719, -6.372, -2151.694]
  MoveL 1198 to (-58.44, 262.16, 260) mm, rotated rx -90 ry -25 rz -51.76 deg; joints [1.97, -46.45, 99.158, 40.084, -108.711, -6.092, -2148.242]
  MoveL 1199 to (-57.77, 266.19, 250) mm, rotated rx -90 ry -25 rz -55.66 deg; joints [1.626, -46.647, 99.516, 39.899, -108.701, -5.814, -2144.344]
  MoveL 1200 to (-56.69, 270.59, 240) mm, rotated rx -90 ry -25 rz -59.96 deg; joints [1.28, -46.843, 99.868, 39.711, -108.687, -5.54, -2140.04]
  MoveL 1201 to (-55.14, 275.28, 230) mm, rotated rx -90 ry -25 rz -64.63 deg; joints [0.933, -47.036, 100.213, 39.52, -108.671, -5.268, -2135.371]
  MoveL 1202 to (-53.04, 280.16, 220) mm, rotated rx -90 ry -25 rz -69.62 deg; joints [0.584, -47.227, 100.551, 39.327, -108.653, -4.998, -2130.377]
  MoveL 1203 to (-50.33, 285.12, 210) mm, rotated rx -90 ry -25 rz -74.91 deg; joints [0.233, -47.414, 100.883, 39.131, -108.633, -4.731, -2125.094]
  MoveL 1204 to (-46.98, 290.04, 200) mm, rotated rx -90 ry -25 rz -80.44 deg; joints [-0.119, -47.598, 101.209, 38.932, -108.611, -4.466, -2119.561]
  MoveL 1205 to (-42.97, 294.79, 190) mm, rotated rx -90 ry -25 rz -86.19 deg; joints [-0.473, -47.778, 101.528, 38.731, -108.588, -4.201, -2113.811]
  MoveL 1206 to (-38.31, 299.24, 180) mm, rotated rx -90 ry -25 rz -92.12 deg; joints [-0.828, -47.955, 101.841, 38.528, -108.564, -3.938, -2107.881]
  MoveL 1207 to (-33.03, 303.26, 170) mm, rotated rx -90 ry -25 rz -98.2 deg; joints [-1.185, -48.126, 102.148, 38.323, -108.539, -3.676, -2101.801]
  MoveL 1208 to (-27.19, 306.74, 160) mm, rotated rx -90 ry -25 rz -104.4 deg; joints [-1.544, -48.292, 102.448, 38.116, -108.514, -3.415, -2095.603]
  MoveL 1209 to (-20.88, 309.56, 150) mm, rotated rx -90 ry -25 rz -110.68 deg; joints [-1.904, -48.453, 102.742, 37.907, -108.49, -3.153, -2089.318]
  MoveL 1210 to (-14.2, 311.65, 140) mm, rotated rx -90 ry -25 rz -117.03 deg; joints [-2.265, -48.609, 103.031, 37.696, -108.465, -2.892, -2082.972]
  MoveL 1211 to (-7.28, 312.93, 130) mm, rotated rx -90 ry -25 rz -123.4 deg; joints [-2.628, -48.758, 103.313, 37.483, -108.442, -2.631, -2076.596]
  MoveL 1212 to (-0.24, 313.38, 120) mm, rotated rx -90 ry -25 rz -129.78 deg; joints [-2.992, -48.902, 103.589, 37.269, -108.419, -2.369, -2070.217]
  MoveL 1213 to (6.77, 312.99, 110) mm, rotated rx -90 ry -25 rz -136.14 deg; joints [-3.358, -49.04, 103.859, 37.053, -108.397, -2.108, -2063.862]
  MoveL 1214 to (13.63, 311.79, 100) mm, rotated rx -90 ry -25 rz -142.44 deg; joints [-3.725, -49.171, 104.123, 36.835, -108.376, -1.846, -2057.558]
  MoveL 1215 to (20.21, 309.81, 90) mm, rotated rx -90 ry -25 rz -148.67 deg; joints [-4.093, -49.297, 104.381, 36.616, -108.356, -1.584, -2051.334]
  MoveL 1216 to (26.38, 307.15, 80) mm, rotated rx -90 ry -25 rz -154.78 deg; joints [-4.463, -49.418, 104.633, 36.395, -108.336, -1.323, -2045.218]
  MoveL 1217 to (32.08, 303.89, 70) mm, rotated rx -90 ry -25 rz -160.76 deg; joints [-4.834, -49.533, 104.879, 36.172, -108.316, -1.062, -2039.241]
  MoveL 1218 to (37.21, 300.16, 60) mm, rotated rx -90 ry -25 rz -166.57 deg; joints [-5.207, -49.643, 105.118, 35.947, -108.296, -0.801, -2033.432]
  MoveL 1219 to (41.73, 296.07, 50) mm, rotated rx -90 ry -25 rz -172.18 deg; joints [-5.581, -49.748, 105.352, 35.72, -108.276, -0.542, -2027.825]
  MoveL 1220 to (45.64, 291.75, 40) mm, rotated rx -90 ry -25 rz -177.55 deg; joints [-5.956, -49.85, 105.579, 35.491, -108.256, -0.284, -2022.451]
  MoveL 1221 to (48.92, 287.33, 30) mm, rotated rx -90 ry -25 rz 177.35 deg; joints [-6.332, -49.947, 105.801, 35.26, -108.234, -0.027, -2017.347]
  MoveL 1222 to (51.6, 282.93, 20) mm, rotated rx -90 ry -25 rz 172.55 deg; joints [-6.709, -50.042, 106.016, 35.028, -108.21, 0.228, -2012.547]
  MoveL 1223 to (53.73, 278.68, 10) mm, rotated rx -90 ry -25 rz 168.09 deg; joints [-7.088, -50.134, 106.224, 34.793, -108.185, 0.482, -2008.09]
  MoveL 1224 to (55.37, 274.67, 0) mm, rotated rx -90 ry -25 rz 164.01 deg; joints [-7.468, -50.223, 106.427, 34.556, -108.158, 0.732, -2004.014]
  Set speed (1000.0 mm/s)
  MoveL 1225 to (55.37, 274.67, 0) mm, rotated rx -90 ry -25 rz 164.01 deg; joints [-7.468, -50.223, 106.427, 34.556, -108.158, 0.732, -2004.014]
  Set speed (1000.0 mm/s)
  MoveL 1226 to (-58.93, 252.99, 290) mm, rotated rx -90 ry -25 rz -42.9 deg; joints [2.992, -45.848, 98.043, 40.621, -108.724, -6.944, -2157.096]
  MoveL 1227 to (-58.93, 252.99, 290) mm, rotated rx -90 ry -25 rz -42.9 deg; joints [2.992, -45.848, 98.043, 40.621, -108.724, -6.944, -2157.096]
  Set speed (60.0 mm/s)
  MoveL 1228 to (-37.11, 208.63, 290) mm, rotated rx -90 ry -25 rz 8.11 deg; joints [2.992, -45.692, 98.056, 40.659, -108.852, -6.827, -2208.107]
  Set speed (1000.0 mm/s)
  MoveL 1229 to (-37.11, 208.63, 290) mm, rotated rx -90 ry -25 rz 8.11 deg; joints [2.992, -45.692, 98.056, 40.659, -108.852, -6.827, -2208.107]
  Set speed (1000.0 mm/s)
  MoveL 1230 to (55.37, 274.67, 0) mm, rotated rx -90 ry -25 rz 164.01 deg; joints [-7.468, -50.223, 106.427, 34.556, -108.158, 0.732, -2364.014]
  MoveL 1231 to (55.37, 274.67, 0) mm, rotated rx -90 ry -25 rz 164.01 deg; joints [-7.468, -50.223, 106.427, 34.556, -108.158, 0.732, -2364.014]
  Set speed (60.0 mm/s)
  MoveL 1232 to (20.49, 309.71, 0) mm, rotated rx -90 ry -25 rz -148.94 deg; joints [-7.468, -50.346, 106.416, 34.531, -108.048, 0.653, -2411.057]
  Set speed (1000.0 mm/s)
  MoveL 1233 to (20.49, 309.71, 0) mm, rotated rx -90 ry -25 rz -148.94 deg; joints [-7.468, -50.346, 106.416, 34.531, -108.048, 0.653, -2411.057]
  Set speed (1000.0 mm/s)
  MoveL 1234 to (55.37, 274.67, 0) mm, rotated rx -90 ry -25 rz 164.01 deg; joints [-7.468, -50.223, 106.427, 34.556, -108.158, 0.732, -2364.014]
  MoveL 1235 to (55.37, 274.67, 0) mm, rotated rx -90 ry -25 rz 164.01 deg; joints [-7.468, -50.223, 106.427, 34.556, -108.158, 0.732, -2364.014]
  Set speed (60.0 mm/s)
  MoveL 1236 to (53.73, 278.68, 10) mm, rotated rx -90 ry -25 rz 168.09 deg; joints [-7.088, -50.134, 106.224, 34.793, -108.185, 0.482, -2368.09]
  MoveL 1237 to (51.6, 282.93, 20) mm, rotated rx -90 ry -25 rz 172.55 deg; joints [-6.709, -50.042, 106.016, 35.028, -108.21, 0.228, -2372.547]
  MoveL 1238 to (48.92, 287.33, 30) mm, rotated rx -90 ry -25 rz 177.35 deg; joints [-6.332, -49.947, 105.801, 35.26, -108.234, -0.027, -2377.347]
  MoveL 1239 to (45.64, 291.75, 40) mm, rotated rx -90 ry -25 rz -177.55 deg; joints [-5.956, -49.85, 105.579, 35.491, -108.256, -0.284, -2382.451]
  MoveL 1240 to (41.73, 296.07, 50) mm, rotated rx -90 ry -25 rz -172.18 deg; joints [-5.581, -49.748, 105.352, 35.72, -108.276, -0.542, -2387.825]
  MoveL 1241 to (37.21, 300.16, 60) mm, rotated rx -90 ry -25 rz -166.57 deg; joints [-5.207, -49.643, 105.118, 35.947, -108.296, -0.801, -2393.432]
  MoveL 1242 to (32.08, 303.89, 70) mm, rotated rx -90 ry -25 rz -160.76 deg; joints [-4.834, -49.533, 104.879, 36.172, -108.316, -1.062, -2399.241]
  MoveL 1243 to (26.38, 307.15, 80) mm, rotated rx -90 ry -25 rz -154.78 deg; joints [-4.463, -49.418, 104.633, 36.395, -108.336, -1.323, -2405.218]
  MoveL 1244 to (20.21, 309.81, 90) mm, rotated rx -90 ry -25 rz -148.67 deg; joints [-4.093, -49.297, 104.381, 36.616, -108.356, -1.584, -2411.334]
  MoveL 1245 to (13.63, 311.79, 100) mm, rotated rx -90 ry -25 rz -142.44 deg; joints [-3.725, -49.171, 104.123, 36.835, -108.376, -1.846, -2417.558]
  MoveL 1246 to (6.77, 312.99, 110) mm, rotated rx -90 ry -25 rz -136.14 deg; joints [-3.358, -49.04, 103.859, 37.053, -108.397, -2.108, -2423.862]
  MoveL 1247 to (-0.24, 313.38, 120) mm, rotated rx -90 ry -25 rz -129.78 deg; joints [-2.992, -48.902, 103.589, 37.269, -108.419, -2.369, -2430.217]
  MoveL 1248 to (-7.28, 312.93, 130) mm, rotated rx -90 ry -25 rz -123.4 deg; joints [-2.628, -48.758, 103.313, 37.483, -108.442, -2.631, -2436.596]
  MoveL 1249 to (-14.2, 311.65, 140) mm, rotated rx -90 ry -25 rz -117.03 deg; joints [-2.265, -48.609, 103.031, 37.696, -108.465, -2.892, -2442.972]
  MoveL 1250 to (-20.88, 309.56, 150) mm, rotated rx -90 ry -25 rz -110.68 deg; joints [-1.904, -48.453, 102.742, 37.907, -108.49, -3.153, -2449.318]
  MoveL 1251 to (-27.19, 306.74, 160) mm, rotated rx -90 ry -25 rz -104.4 deg; joints [-1.544, -48.292, 102.448, 38.116, -108.514, -3.415, -2455.603]
  MoveL 1252 to (-33.03, 303.26, 170) mm, rotated rx -90 ry -25 rz -98.2 deg; joints [-1.185, -48.126, 102.148, 38.323, -108.539, -3.676, -2461.801]
  MoveL 1253 to (-38.31, 299.24, 180) mm, rotated rx -90 ry -25 rz -92.12 deg; joints [-0.828, -47.955, 101.841, 38.528, -108.564, -3.938, -2467.881]
  MoveL 1254 to (-42.97, 294.79, 190) mm, rotated rx -90 ry -25 rz -86.19 deg; joints [-0.473, -47.778, 101.528, 38.731, -108.588, -4.201, -2473.811]
  MoveL 1255 to (-46.98, 290.04, 200) mm, rotated rx -90 ry -25 rz -80.44 deg; joints [-0.119, -47.598, 101.209, 38.932, -108.611, -4.466, -2479.561]
  MoveL 1256 to (-50.33, 285.12, 210) mm, rotated rx -90 ry -25 rz -74.91 deg; joints [0.233, -47.414, 100.883, 39.131, -108.633, -4.731, -2485.094]
  MoveL 1257 to (-53.04, 280.16, 220) mm, rotated rx -90 ry -25 rz -69.62 deg; joints [0.584, -47.227, 100.551, 39.327, -108.653, -4.998, -2490.377]
  MoveL 1258 to (-55.14, 275.28, 230) mm, rotated rx -90 ry -25 rz -64.63 deg; joints [0.933, -47.036, 100.213, 39.52, -108.671, -5.268, -2495.371]
  MoveL 1259 to (-56.69, 270.59, 240) mm, rotated rx -90 ry -25 rz -59.96 deg; joints [1.28, -46.843, 99.868, 39.711, -108.687, -5.54, -2500.04]
  MoveL 1260 to (-57.77, 266.19, 250) mm, rotated rx -90 ry -25 rz -55.66 deg; joints [1.626, -46.647, 99.516, 39.899, -108.701, -5.814, -2504.344]
  MoveL 1261 to (-58.44, 262.16, 260) mm, rotated rx -90 ry -25 rz -51.76 deg; joints [1.97, -46.45, 99.158, 40.084, -108.711, -6.092, -2508.242]
  MoveL 1262 to (-58.8, 258.59, 270) mm, rotated rx -90 ry -25 rz -48.31 deg; joints [2.312, -46.251, 98.793, 40.266, -108.719, -6.372, -2511.694]
  MoveL 1263 to (-58.94, 255.51, 280) mm, rotated rx -90 ry -25 rz -45.34 deg; joints [2.653, -46.05, 98.421, 40.445, -108.723, -6.656, -2514.659]
  MoveL 1264 to (-58.93, 252.99, 290) mm, rotated rx -90 ry -25 rz -42.9 deg; joints [2.992, -45.848, 98.043, 40.621, -108.724, -6.944, -2517.096]
  Set speed (1000.0 mm/s)
  MoveL 1265 to (-58.93, 252.99, 290) mm, rotated rx -90 ry -25 rz -42.9 deg; joints [2.992, -45.848, 98.043, 40.621, -108.724, -6.944, -2517.096]
  Set speed (1000.0 mm/s)
  MoveL 1266 to (-37.11, 208.63, 290) mm, rotated rx -90 ry -25 rz 8.11 deg; joints [2.992, -45.692, 98.056, 40.659, -108.852, -6.827, -2568.107]
  MoveL 1267 to (-37.11, 208.63, 290) mm, rotated rx -90 ry -25 rz 8.11 deg; joints [2.992, -45.692, 98.056, 40.659, -108.852, -6.827, -2568.107]
  Set speed (60.0 mm/s)
  MoveL 1268 to (-39.03, 210.26, 280) mm, rotated rx -90 ry -25 rz 5.51 deg; joints [2.653, -45.891, 98.435, 40.483, -108.854, -6.538, -2565.515]
  MoveL 1269 to (-41.29, 212.35, 270) mm, rotated rx -90 ry -25 rz 2.36 deg; joints [2.312, -46.089, 98.807, 40.305, -108.853, -6.252, -2562.358]
  MoveL 1270 to (-43.78, 214.95, 260) mm, rotated rx -90 ry -25 rz -1.32 deg; joints [1.97, -46.284, 99.173, 40.123, -108.849, -5.969, -2558.681]
  MoveL 1271 to (-46.4, 218.08, 250) mm, rotated rx -90 ry -25 rz -5.47 deg; joints [1.626, -46.479, 99.531, 39.939, -108.841, -5.69, -2554.527]
  MoveL 1272 to (-49.06, 221.75, 240) mm, rotated rx -90 ry -25 rz -10.06 deg; joints [1.28, -46.672, 99.883, 39.751, -108.83, -5.414, -2549.94]
  MoveL 1273 to (-51.62, 225.97, 230) mm, rotated rx -90 ry -25 rz -15.04 deg; joints [0.933, -46.864, 100.228, 39.56, -108.815, -5.142, -2544.964]
  MoveL 1274 to (-53.98, 230.73, 220) mm, rotated rx -90 ry -25 rz -20.35 deg; joints [0.584, -47.055, 100.567, 39.367, -108.797, -4.873, -2539.646]
  MoveL 1275 to (-56, 236.01, 210) mm, rotated rx -90 ry -25 rz -25.97 deg; joints [0.233, -47.244, 100.899, 39.17, -108.776, -4.608, -2534.028]
  MoveL 1276 to (-57.57, 241.75, 200) mm, rotated rx -90 ry -25 rz -31.84 deg; joints [-0.119, -47.432, 101.224, 38.971, -108.752, -4.345, -2528.155]
  MoveL 1277 to (-58.59, 247.88, 190) mm, rotated rx -90 ry -25 rz -37.93 deg; joints [-0.473, -47.618, 101.543, 38.768, -108.724, -4.086, -2522.068]
  MoveL 1278 to (-58.95, 254.32, 180) mm, rotated rx -90 ry -25 rz -44.19 deg; joints [-0.828, -47.801, 101.855, 38.563, -108.694, -3.828, -2515.809]
  MoveL 1279 to (-58.59, 260.95, 170) mm, rotated rx -90 ry -25 rz -50.58 deg; joints [-1.185, -47.982, 102.161, 38.356, -108.662, -3.573, -2509.416]
  MoveL 1280 to (-57.45, 267.65, 160) mm, rotated rx -90 ry -25 rz -57.07 deg; joints [-1.544, -48.16, 102.46, 38.146, -108.628, -3.32, -2502.926]
  MoveL 1281 to (-55.51, 274.28, 150) mm, rotated rx -90 ry -25 rz -63.63 deg; joints [-1.904, -48.334, 102.753, 37.934, -108.592, -3.069, -2496.375]
  MoveL 1282 to (-52.77, 280.72, 140) mm, rotated rx -90 ry -25 rz -70.2 deg; joints [-2.265, -48.505, 103.04, 37.719, -108.556, -2.819, -2489.796]
  MoveL 1283 to (-49.26, 286.82, 130) mm, rotated rx -90 ry -25 rz -76.78 deg; joints [-2.628, -48.671, 103.321, 37.503, -108.518, -2.569, -2483.221]
  MoveL 1284 to (-45.04, 292.47, 120) mm, rotated rx -90 ry -25 rz -83.32 deg; joints [-2.992, -48.832, 103.595, 37.285, -108.48, -2.32, -2476.68]
  MoveL 1285 to (-40.19, 297.56, 110) mm, rotated rx -90 ry -25 rz -89.8 deg; joints [-3.358, -48.988, 103.864, 37.064, -108.442, -2.072, -2470.201]
  MoveL 1286 to (-34.83, 302, 100) mm, rotated rx -90 ry -25 rz -96.19 deg; joints [-3.725, -49.138, 104.126, 36.842, -108.405, -1.823, -2463.814]
  MoveL 1287 to (-29.06, 305.72, 90) mm, rotated rx -90 ry -25 rz -102.46 deg; joints [-4.093, -49.283, 104.382, 36.619, -108.368, -1.575, -2457.545]
  MoveL 1288 to (-23.03, 308.7, 80) mm, rotated rx -90 ry -25 rz -108.58 deg; joints [-4.463, -49.423, 104.632, 36.393, -108.331, -1.327, -2451.421]
  MoveL 1289 to (-16.86, 310.92, 70) mm, rotated rx -90 ry -25 rz -114.53 deg; joints [-4.834, -49.556, 104.876, 36.166, -108.295, -1.078, -2445.47]
  MoveL 1290 to (-10.69, 312.41, 60) mm, rotated rx -90 ry -25 rz -120.28 deg; joints [-5.207, -49.684, 105.115, 35.938, -108.259, -0.83, -2439.72]
  MoveL 1291 to (-4.64, 313.2, 50) mm, rotated rx -90 ry -25 rz -125.8 deg; joints [-5.581, -49.807, 105.347, 35.708, -108.224, -0.581, -2434.198]
  MoveL 1292 to (1.18, 313.37, 40) mm, rotated rx -90 ry -25 rz -131.07 deg; joints [-5.956, -49.924, 105.573, 35.476, -108.19, -0.333, -2428.933]
  MoveL 1293 to (6.67, 313.01, 30) mm, rotated rx -90 ry -25 rz -136.04 deg; joints [-6.332, -50.036, 105.793, 35.242, -108.155, -0.085, -2423.955]
  MoveL 1294 to (11.76, 312.2, 20) mm, rotated rx -90 ry -25 rz -140.7 deg; joints [-6.709, -50.143, 106.006, 35.007, -108.12, 0.162, -2419.296]
  MoveL 1295 to (16.38, 311.06, 10) mm, rotated rx -90 ry -25 rz -145.01 deg; joints [-7.088, -50.246, 106.214, 34.77, -108.084, 0.408, -2414.985]
  MoveL 1296 to (20.49, 309.71, 0) mm, rotated rx -90 ry -25 rz -148.94 deg; joints [-7.468, -50.346, 106.416, 34.531, -108.048, 0.653, -2411.057]
  Set speed (1000.0 mm/s)
  MoveL 1297 to (20.49, 309.71, 0) mm, rotated rx -90 ry -25 rz -148.94 deg; joints [-7.468, -50.346, 106.416, 34.531, -108.048, 0.653, -2411.057]
  Set speed (1000.0 mm/s)
  MoveL 1298 to (-37.11, 208.63, 290) mm, rotated rx -90 ry -25 rz 8.11 deg; joints [2.992, -45.692, 98.056, 40.659, -108.852, -6.827, -2568.107]
  MoveL 1299 to (-37.11, 208.63, 290) mm, rotated rx -90 ry -25 rz 8.11 deg; joints [2.992, -45.692, 98.056, 40.659, -108.852, -6.827, -2568.107]
  Set speed (60.0 mm/s)
  MoveL 1300 to (-43.85, 188.95, 290) mm, rotated rx -90 ry -25 rz 14.31 deg; joints [2.992, -46.574, 97.966, 40.447, -108.114, -7.494, -2574.314]
  Set speed (1000.0 mm/s)
  MoveL 1301 to (-43.85, 188.95, 290) mm, rotated rx -90 ry -25 rz 14.31 deg; joints [2.992, -46.574, 97.966, 40.447, -108.114, -7.494, -2574.314]
  Set speed (1000.0 mm/s)
  MoveL 1302 to (20.49, 309.71, 0) mm, rotated rx -90 ry -25 rz -148.94 deg; joints [-7.468, -50.346, 106.416, 34.531, -108.048, 0.653, -2411.057]
